//   DUTs/IO/Topology/ Beckhoff_AMI8xxxEK1122_B38FD36B.TcDUT (not stored), EK1100_Beckhoff_AMI8xxx_4205BDB3.TcDUT (not stored), EtherCAT_Master_AMIxxxx_FECF87C2.TcDUT (not stored), Beckhoff_APS1xxxEK1122_85E711A3.TcDUT (not stored), Beckhoff_APS1xxx_0455F8D3.TcDUT (not stored), Beckhoff_APS4xxxEK1122_65CE088F.TcDUT (not stored), Beckhoff_APS4xxx_87463DAF.TcDUT (not stored), EtherCAT_Master_APSxxxx_6FACD001.TcDUT (not stored), A_0060_AT2020_0250_0019_AT2020_0250_DEA07AF9.TcDUT (not stored), A_0036_AT2040_0250_0021_A3885EBC.TcDUT (not stored), A_0037_AT2040_0250_0022_971D272D.TcDUT (not stored), A_0038_AT2040_0250_0023_2AEAC7B2.TcDUT (not stored), A_0039_AT2040_0250_0024_A0FBBBF9.TcDUT (not stored), A_0040_AT2041_0250_0018_599416E0.TcDUT (not stored), A_0041_AT2041_0250_0019_45B99D70.TcDUT (not stored), A_0042_AT2041_0250_0020_B304CC62.TcDUT (not stored), A_0043_AT2041_0250_0021_3915B029.TcDUT (not stored), A_0044_AT2041_0250_0022_EA8B7A1C.TcDUT (not stored), A_0045_AT2041_0250_0023_5C753B73.TcDUT (not stored), A_0046_AT2042_0250_0024_35EBD522.TcDUT (not stored), A_0047_AT2050_0500_0016_017EACB3.TcDUT (not stored), A_0048_AT2050_0500_0017_A8B58F1D.TcDUT (not stored), A_0049_AT2050_0500_0018_A5979C2D.TcDUT (not stored), A_0050_AT2050_0500_0019_E6F81550.TcDUT (not stored), A_0051_AT2050_0500_0020_6A24DD88.TcDUT (not stored), A_0052_AT2050_0500_0021_294B54F5.TcDUT (not stored), A_0053_AT2050_0500_0022_49FE826D.TcDUT (not stored), A_0054_AT2050_0500_0023_9DD4EAFB.TcDUT (not stored), A_0055_AT2050_0500_0024_F6D8BACC.TcDUT (not stored), A_0056_AT2050_0501_0017_5F139962.TcDUT (not stored), A_0057_AT2050_0501_0020_6B86E0F3.TcDUT (not stored), A_0058_AT2050_0501_0021_54B106B2.TcDUT (not stored), A_0061_AT2020_0250_0023_AT2020_0250_0F2EDFD4.TcDUT (not stored), A_0062_AT2025_0250_0020_AT2025_0250_13035444.TcDUT (not stored), A_0063_AT2025_0250_0022_AT2025_0250_9D18840C.TcDUT (not stored), A_0064_AT2025_0250_0023_AT2025_0250_4A8CE23A.TcDUT (not stored), A_0065_AT2026_0250_0019_AT2026_0250_E347C194.TcDUT (not stored), A_0066_AT2026_0250_0020_AT2026_0250_D7D2B805.TcDUT (not stored), A_0067_AT2026_0250_0022_AT2026_0250_D02FEC70.TcDUT (not stored), A_0068_AT2026_0250_0024_AT2026_0250_BF201DA5.TcDUT (not stored), A_0069_AT2050_0501_0019_AT2050_0501_0D0F91BF.TcDUT (not stored), A_0070_AT2050_0501_0022_AT2050_0501_871EEDF4.TcDUT (not stored), A_0071_AT2050_0501_0023_AT2050_0501_6B46D2C7.TcDUT (not stored), A_0072_AT2050_0501_0024_AT2050_0501_776B5957.TcDUT (not stored), Beckhoff_AT2xxxEK1122_56C52038.TcDUT (not stored), Beckhoff_AT1xxx_7510A45A.TcDUT (not stored), A_0001_ATH2000_0250_0022_20236C4E.TcDUT (not stored), A_0002_ATH2000_0250_0023_D700A2ED.TcDUT (not stored), Beckhoff_ATH2xxxEK1122_13FBDC00.TcDUT (not stored), Beckhoff_ATH2xxx_159CB27D.TcDUT (not stored), EtherCAT_Master_ATxxxx_83672136.TcDUT (not stored), Beckhoff_AX2xxxEK1122_5FAF3C40.TcDUT (not stored), Beckhoff_AX2xxx_B0467A4D.TcDUT (not stored), Beckhoff_AX5xxxEK1122_5EFAAD43.TcDUT (not stored), Beckhoff_AX5xxx_ABA3CB51.TcDUT (not stored), Beckhoff_AX8yxxEK1122_5DB842B3.TcDUT (not stored), Beckhoff_AX8yxx_9373B1FA.TcDUT (not stored), Beckhoff_AX86xxEK1122_9E61CBD7.TcDUT (not stored), Beckhoff_AX86xx_1E3C21C9.TcDUT (not stored), Beckhoff_AX88xxEK1122_27E1F918.TcDUT (not stored), Beckhoff_AX88xx_5781E6BD.TcDUT (not stored), EtherCAT_Master_AXxxxx_5BD89A80.TcDUT (not stored), A_0014_BK1250_0000_0000_A4796D49.TcDUT (not stored), Beckhoff_BKxxxxsub_EK1100_CE1F4926.TcDUT (not stored), A_0001_BK1120_0000_0000_A11D37A6.TcDUT (not stored), A_0002_BK1120_0000_0001_6C916313.TcDUT (not stored), A_0003_BK1120_0000_0016_3EC4837B.TcDUT (not stored), A_0004_BK1120_0000_0017_F348D7CE.TcDUT (not stored), A_0005_BK1120_0000_0018_EC8BABB1.TcDUT (not stored), A_0006_BK1120_0000_0019_2107FF04.TcDUT (not stored), A_0007_BK1120_0000_0020_2D4D5A66.TcDUT (not stored), A_0008_BK1120_0000_0021_E0C10ED3.TcDUT (not stored), A_0009_CPXXXX_BK1150_0016_B294EEBB.TcDUT (not stored), A_0010_BK1150_0000_0016_7F18BA0E.TcDUT (not stored), A_0011_BK1150_0000_0017_163F2E6B.TcDUT (not stored), A_0012_BK1150_0000_0018_DBB37ADE.TcDUT (not stored), A_0013_BK1150_0000_0019_89E69AB6.TcDUT (not stored), A_0016_BK1250_0000_0017_446ACE03.TcDUT (not stored), Term_474_EK1100_44DC070B.TcDUT (not stored), A_0018_BK1250_0000_0019_5BA9B27C.TcDUT (not stored), Term_476_EK1100_ED4AD6ED.TcDUT (not stored), A_0017_BK1250_0000_0018_9625E6C9.TcDUT (not stored), Term_478_EK1100_69E708A2.TcDUT (not stored), A_0019_IL2300_B110_0016_D7C567E6.TcDUT (not stored), A_0020_IL2300_B110_0017_5C3C5D52.TcDUT (not stored), A_0021_IL2301_B110_0016_18E5DAA8.TcDUT (not stored), A_0022_IL2301_B110_0017_CE2B414F.TcDUT (not stored), A_0023_IL2302_B110_0016_9156D55C.TcDUT (not stored), A_0024_IL2302_B110_0017_7CD378DF.TcDUT (not stored), Beckhoff_BKxxxxEK1122_F2DB5C09.TcDUT (not stored), A_0015_BK1250_0000_0016_69F539FC.TcDUT (not stored), Beckhoff_BKxxxx_655B2331.TcDUT (not stored), A_0006_CU1128_0000_0002_0DB5F5B9.TcDUT (not stored), A_0005_CU1128_0000_0001_15602991.TcDUT (not stored), A_0004_CU1128_0000_0000_E069C544.TcDUT (not stored), A_0003_CU1124_0000_0016_F6CF179A.TcDUT (not stored), A_0002_CU1123_0010_0016_C16CD0B3.TcDUT (not stored), A_0001_CU1123_0000_0016_A8E4CC63.TcDUT (not stored), Beckhoff_CUxxxxEK1122_8084EAF6.TcDUT (not stored), Beckhoff_CUxxxx_D57B3A25.TcDUT (not stored), Beckhoff_CXxxxxEK1122_6E1B70A9.TcDUT (not stored), Beckhoff_CXxxxx_5AB893DE.TcDUT (not stored), TcTerminals210_1BK1250_5A51D777.TcDUT (not stored), TcTerminals210_EK1100_1_99191ECD.TcDUT (not stored), TcTerminals210_2BK1250_08988889.TcDUT (not stored), TcTerminals210_EK1100_2_BDAFA3B6.TcDUT (not stored), EtherCAT_Master_BKCUCX_8F70BCEA.TcDUT (not stored), Beckhoff_EJ1xxxEK1122_5D41058A.TcDUT (not stored), Beckhoff_EJ1xxx_BA4DEDCC.TcDUT (not stored), Beckhoff_EJ2xxxEK1122_7BCCD4D9.TcDUT (not stored), Beckhoff_EJ2xxx_42F4B05B.TcDUT (not stored), Beckhoff_EJ3xxxEK1122_6922078E.TcDUT (not stored), Beckhoff_EJ3xxx_E0C24C98.TcDUT (not stored), Beckhoff_EJ4xxxEK1122_15AA3F2B.TcDUT (not stored), Beckhoff_EJ4xxx_B433EAC7.TcDUT (not stored), Beckhoff_EJ5xxxEK1122_0744EC7C.TcDUT (not stored), Beckhoff_EJ5xxx_DF22D5A3.TcDUT (not stored), Beckhoff_EJ6xxxEK1122_30779985.TcDUT (not stored), Beckhoff_EJ6xxx_A0E5C2C0.TcDUT (not stored), Beckhoff_EJ7xxxEK1122_22994AD2.TcDUT (not stored), Beckhoff_EJ7xxx_9F75012E.TcDUT (not stored), Beckhoff_EJ9xxxEK1122_DB893B98.TcDUT (not stored), Beckhoff_EJ9xxx_660B2C8D.TcDUT (not stored), Beckhoff_EJx9xxEK1122_05D2B413.TcDUT (not stored), Beckhoff_EJx9xx_A9128509.TcDUT (not stored), EtherCAT_Master_EJxxxx_A1D13F1B.TcDUT (not stored), Beckhoff_EK11xxEK1122_0F9A1885.TcDUT (not stored), Beckhoff_EK11xx_C12453FF.TcDUT (not stored), Beckhoff_EK12xxEK1122_E9998301.TcDUT (not stored), Beckhoff_EK12xx_26FD3E4A.TcDUT (not stored), Beckhoff_EK13xxEK1122_7883D180.TcDUT (not stored), Beckhoff_EK13xx_F78FC0F8.TcDUT (not stored), Beckhoff_EK15xxEK1122_F4825052.TcDUT (not stored), Beckhoff_EK15xx_2CCE234B.TcDUT (not stored), Beckhoff_EK18xxEK1122_46BB19D8.TcDUT (not stored), Beckhoff_EK18xx_2BB31392.TcDUT (not stored), Beckhoff_EKM1xxxEK1122_D80A806C.TcDUT (not stored), Beckhoff_EKM1xxx_4291A3D4.TcDUT (not stored), Beckhoff_EKx9xxEK1122_199990A5.TcDUT (not stored), Beckhoff_EKx9xx_14304971.TcDUT (not stored), Beckhoff_EKxxxx_0080EK1122_49C116CC.TcDUT (not stored), Beckhoff_EKxxxx_0080_F8E2E0BC.TcDUT (not stored), EtherCAT_Master_EKxxxx_AFFC15C4.TcDUT (not stored), Beckhoff_ELM3xxxEK1122_52A3E13B.TcDUT (not stored), Beckhoff_ELM3xxx_6EC4C133.TcDUT (not stored), Beckhoff_ELM31xxEK1122_3E17608C.TcDUT (not stored), Beckhoff_ELM31xx_1B5DD775.TcDUT (not stored), Beckhoff_ELM35xxEK1122_B82F516C.TcDUT (not stored), Beckhoff_ELM35xx_45F1AC79.TcDUT (not stored), Beckhoff_ELM36xxEK1122_DABD45E4.TcDUT (not stored), Beckhoff_ELM36xx_F5043D7C.TcDUT (not stored), Beckhoff_ELM37xxEK1122_FB33499C.TcDUT (not stored), Beckhoff_ELM37xx_37DB7D9A.TcDUT (not stored), Beckhoff_ELM3xxx_0030EK1122_7F195F23.TcDUT (not stored), Beckhoff_ELM3xxx_0030_86EC0720.TcDUT (not stored), Beckhoff_ELM9xxxEK1122_E008DD2D.TcDUT (not stored), Beckhoff_ELM9xxx_2CCFEFDC.TcDUT (not stored), EtherCAT_Master_ELMxxxx_F3377F79.TcDUT (not stored), Beckhoff_EL1xxxEK1122_BA3F35BD.TcDUT (not stored), Beckhoff_EL1xxx_A02C084E.TcDUT (not stored), Beckhoff_EL2xxxEK1122_8D0C4044.TcDUT (not stored), Beckhoff_EL2xxx_6D51086F.TcDUT (not stored), Beckhoff_EL3xxxEK1122_9FE29313.TcDUT (not stored), Beckhoff_EL3xxx_68884AC1.TcDUT (not stored), Beckhoff_EL3xxx_0030EK1122_A8C7E601.TcDUT (not stored), Beckhoff_EL3xxx_0030_2D07FB6C.TcDUT (not stored), Beckhoff_EL4xxxEK1122_E36AABB6.TcDUT (not stored), Beckhoff_EL4xxx_B43A2050.TcDUT (not stored), Beckhoff_EL5xxxEK1122_F18478E1.TcDUT (not stored), Beckhoff_EL5xxx_C80BAEFE.TcDUT (not stored), Beckhoff_EL6xxxEK1122_C6B70D18.TcDUT (not stored), Beckhoff_EL6xxx_F14D3E2E.TcDUT (not stored), Beckhoff_EL7xxxEK1122_D459DE4F.TcDUT (not stored), Beckhoff_EL7xxx_9130E37B.TcDUT (not stored), Beckhoff_EL9xxxEK1122_2D49AF05.TcDUT (not stored), Beckhoff_EL9xxx_842928EF.TcDUT (not stored), Beckhoff_EL15xxEK1122_50B385EA.TcDUT (not stored), Beckhoff_EL15xx_DB59F57A.TcDUT (not stored), Beckhoff_EL19xxEK1122_DE3ACA7D.TcDUT (not stored), Beckhoff_EL19xx_39A0946F.TcDUT (not stored), Beckhoff_EL25xxEK1122_6780F013.TcDUT (not stored), Beckhoff_EL25xx_19393863.TcDUT (not stored), Beckhoff_EL29xxEK1122_E909BF84.TcDUT (not stored), Beckhoff_EL29xx_4C00A64E.TcDUT (not stored), Beckhoff_EL30xxEK1122_D2D81EDC.TcDUT (not stored), Beckhoff_EL30xx_21D80093.TcDUT (not stored), Beckhoff_EL31xxEK1122_F35612A4.TcDUT (not stored), Beckhoff_EL31xx_0F318B7E.TcDUT (not stored), Beckhoff_EL32xxEK1122_91C4062C.TcDUT (not stored), Beckhoff_EL32xx_64999344.TcDUT (not stored), Beckhoff_EL33xxEK1122_B04A0A54.TcDUT (not stored), Beckhoff_EL33xx_B84F5D38.TcDUT (not stored), Beckhoff_EL34xxEK1122_54E02F3C.TcDUT (not stored), Beckhoff_EL34xx_4C2EC3D0.TcDUT (not stored), Beckhoff_EL37xxEK1122_36723BB4.TcDUT (not stored), Beckhoff_EL37xx_735867E2.TcDUT (not stored), Beckhoff_EL47xxEK1122_4AFA0311.TcDUT (not stored), Beckhoff_EL47xx_965E5194.TcDUT (not stored), Beckhoff_EL66xxEK1122_D63A030B.TcDUT (not stored), Beckhoff_EL66xx_C1E1F370.TcDUT (not stored), Beckhoff_EL67xxEK1122_6F27A5BF.TcDUT (not stored), Beckhoff_EL67xx_2DE66D45.TcDUT (not stored), Beckhoff_EL68xxEK1122_833CFEA0.TcDUT (not stored), Beckhoff_EL68xx_2DEB682D.TcDUT (not stored), Beckhoff_EL69xxEK1122_A2B2F2D8.TcDUT (not stored), Beckhoff_EL69xx_A41E2827.TcDUT (not stored), Beckhoff_EL72xxEK1122_DA7F4B70.TcDUT (not stored), Beckhoff_EL72xx_B1894506.TcDUT (not stored), Beckhoff_EL73xxEK1122_FBF14708.TcDUT (not stored), Beckhoff_EL73xx_9CF0DC04.TcDUT (not stored), Beckhoff_EL99xxEK1122_494C50C5.TcDUT (not stored), A_0003_EL9930_0000_0017_255119B7.TcDUT (not stored), A_0001_EL9930_0000_0016_8200DBB0.TcDUT (not stored), Beckhoff_EL99xx_E89A1FE1.TcDUT (not stored), EtherCAT_Master_ELxxxx_D51EE2EF.TcDUT (not stored), Beckhoff_ELXxxxxEK1122_CE175A58.TcDUT (not stored), Beckhoff_ELXxxxx_091FCA88.TcDUT (not stored), EtherCAT_Master_ELXxxxx_037A66B5.TcDUT (not stored), Beckhoff_EM2xxxEK1122_264CF75A.TcDUT (not stored), Beckhoff_EM2xxx_D8CD5456.TcDUT (not stored), Beckhoff_EM3xxxEK1122_34A2240D.TcDUT (not stored), Beckhoff_EM3xxx_0E1B0655.TcDUT (not stored), Beckhoff_EM7xxxEK1122_7F196951.TcDUT (not stored), Beckhoff_EM7xxx_B71DC934.TcDUT (not stored), EtherCAT_Master_EMxxxx_4F6AEAF3.TcDUT (not stored), A_0024_EPP1342_0001_0017_B861A008.TcDUT (not stored), A_0023_EPP1342_0001_0016_F32E5EF0.TcDUT (not stored), A_0022_EPP1332_0001_0017_4E5F00D5.TcDUT (not stored), A_0021_EPP1332_0001_0016_0C75CF60.TcDUT (not stored), A_0020_EPP1322_0001_0017_AE45DA7A.TcDUT (not stored), A_0019_EPP1322_0001_0016_1D230593.TcDUT (not stored), A_0018_EPP1321_0060_0016_CF61AE2B.TcDUT (not stored), Beckhoff_EPP1xxxEK1122_CF9B9B85.TcDUT (not stored), Beckhoff_EPP1xxx_9DC54301.TcDUT (not stored), Beckhoff_EPP2xxxEK1122_0CAC7812.TcDUT (not stored), Beckhoff_EPP2xxx_7FE046AD.TcDUT (not stored), Beckhoff_EPP3xxxEK1122_936585F9.TcDUT (not stored), Beckhoff_EPP3xxx_5AF4C5F1.TcDUT (not stored), Beckhoff_EPP4xxxEK1122_A96F30AF.TcDUT (not stored), Beckhoff_EPP4xxx_454DDD33.TcDUT (not stored), Beckhoff_EPP5xxxEK1122_277DA9AB.TcDUT (not stored), Beckhoff_EPP5xxx_36D2ADAB.TcDUT (not stored), Beckhoff_EPP6xxxEK1122_580439A8.TcDUT (not stored), Beckhoff_EPP6xxx_5B035970.TcDUT (not stored), Beckhoff_EPP7xxxEK1122_0D11CA3B.TcDUT (not stored), Beckhoff_EPP7xxx_19C1DAAF.TcDUT (not stored), Beckhoff_EPP9xxxEK1122_5167694C.TcDUT (not stored), Beckhoff_EPP9xxx_B13825D2.TcDUT (not stored), EtherCAT_Master_EPPxxxx_7CC0E3EC.TcDUT (not stored), A_0037_EP1312_0001_0016_91E425AA.TcDUT (not stored), A_0026_EP1122_0001_0018_C0E43096.TcDUT (not stored), A_0025_EP1122_0001_0017_02B37791.TcDUT (not stored), A_0024_EP1122_0001_0016_1C40CD3A.TcDUT (not stored), Beckhoff_EP1xxxEK1122_B7B20563.TcDUT (not stored), Beckhoff_EP1xxx_C8E7C95B.TcDUT (not stored), Beckhoff_EP2xxxEK1122_CF43FCA1.TcDUT (not stored), Beckhoff_EP2xxx_B2F46B5A.TcDUT (not stored), Beckhoff_EP3xxxEK1122_961F7095.TcDUT (not stored), Beckhoff_EP3xxx_2B029919.TcDUT (not stored), Beckhoff_EP4xxxEK1122_BB643D5B.TcDUT (not stored), Beckhoff_EP4xxx_3DB4D53F.TcDUT (not stored), Beckhoff_EP5xxxEK1122_41313438.TcDUT (not stored), Beckhoff_EP5xxx_8FA7D670.TcDUT (not stored), Beckhoff_EP6xxxEK1122_E79FCD0D.TcDUT (not stored), Beckhoff_EP6xxx_66B3A0F3.TcDUT (not stored), A_0054_EP7402_0057_0017_54490F59.TcDUT (not stored), Beckhoff_EP7xxxEK1122_A7CCCB3C.TcDUT (not stored), Beckhoff_EP7xxx_5B32BB7C.TcDUT (not stored), Beckhoff_EP8xxxEK1122_09026D55.TcDUT (not stored), Beckhoff_EP8xxx_A1F98A04.TcDUT (not stored), A_0024_EP9521_0020_0000_2C408F2A.TcDUT (not stored), A_0022_EP9224_0037_0017_E33DE408.TcDUT (not stored), A_0013_EP9128_0021_0019_07EDD1EA.TcDUT (not stored), A_0010_EP9128_0021_0018_A4E84267.TcDUT (not stored), A_0007_EP9128_0021_0017_0A93B569.TcDUT (not stored), A_0004_EP9128_0021_0016_B7B89D3D.TcDUT (not stored), A_0001_EP9128_0020_0016_7FD3BAFD.TcDUT (not stored), Beckhoff_EP9xxxEK1122_D439D8FD.TcDUT (not stored), Beckhoff_EP9xxx_40638FD6.TcDUT (not stored), EtherCAT_Master_EPxxxx_AD623DA0.TcDUT (not stored), Beckhoff_EQ1xxxEK1122_FDDE2AD8.TcDUT (not stored), Beckhoff_EQ1xxx_822DEADB.TcDUT (not stored), Beckhoff_EQ2xxxEK1122_609ED827.TcDUT (not stored), Beckhoff_EQ2xxx_ABA09D4F.TcDUT (not stored), Beckhoff_EQ3xxxEK1122_C2B88B71.TcDUT (not stored), Beckhoff_EQ3xxx_1BCF419C.TcDUT (not stored), EtherCAT_Master_EQxxxx_C1E8A49A.TcDUT (not stored), Beckhoff_ER1xxxEK1122_03B27612.TcDUT (not stored), Beckhoff_ER1xxx_F144525A.TcDUT (not stored), Beckhoff_ER2xxxEK1122_C26931CF.TcDUT (not stored), Beckhoff_ER2xxx_C2CD7B25.TcDUT (not stored), Beckhoff_ER3xxxEK1122_1C34A142.TcDUT (not stored), Beckhoff_ER3xxx_0B6E7FA9.TcDUT (not stored), Beckhoff_ER4xxxEK1122_D1435FD1.TcDUT (not stored), Beckhoff_ER4xxx_C7805EB0.TcDUT (not stored), Beckhoff_ER5xxxEK1122_8A557ABF.TcDUT (not stored), Beckhoff_ER5xxx_1B1665E3.TcDUT (not stored), Beckhoff_ER6xxxEK1122_7ED5D873.TcDUT (not stored), Beckhoff_ER6xxx_39EF444F.TcDUT (not stored), Beckhoff_ER7xxxEK1122_C27AB41B.TcDUT (not stored), Beckhoff_ER7xxx_A258BD7D.TcDUT (not stored), Beckhoff_ER8xxxEK1122_05C4D0D1.TcDUT (not stored), Beckhoff_ER8xxx_BCCF5157.TcDUT (not stored), EtherCAT_Master_ERxxxx_D3400E61.TcDUT (not stored), TcTerminals210_1EK1100_99191ECD.TcDUT (not stored), TcTerminals210_2EK1100_BDAFA3B6.TcDUT (not stored), EtherCAT_Master_KLxxxx_4E9397D5.TcDUT (not stored), EtherCAT_Master_KLxxxx_1_B89C6D7A.TcDUT (not stored), EtherCAT_Master_KLxxxx_2_C1BBE75B.TcDUT (not stored), boxesEK1122_6347E441.TcDUT (not stored), boxes_B14E9406.TcDUT (not stored), EtherCAT_Master_Duplicates_FF3295D1.TcDUT (not stored)
//   GVLs/ GVL_iXlinker.TcGVL

// ---- DUTs/IO/Boxes/EK1100_179A0949.TcDUT
{attribute addProperty BoxType "EK1100-0000-0018"}
{attribute addProperty Id "InfoDataInfoData_192954DE162"}
{attribute addProperty CRC "395970889"}
{attribute addProperty SizeInBites "16"}
{attribute addProperty SizeInBytes "2"}
TYPE EK1100_179A0949 :
STRUCT
	{attribute addProperty Name "InfoData"}
	InfoData : InfoData_192954DE;
END_STRUCT
END_TYPE

// ---- DUTs/IO/Boxes/EK1122_179A0949.TcDUT
{attribute addProperty BoxType "EK1122-0000-0018"}
{attribute addProperty Id "InfoDataInfoData_192954DE162"}
{attribute addProperty CRC "395970889"}
{attribute addProperty SizeInBites "16"}
{attribute addProperty SizeInBytes "2"}
TYPE EK1122_179A0949 :
STRUCT
	{attribute addProperty Name "InfoData"}
	InfoData : InfoData_192954DE;
END_STRUCT
END_TYPE

// ---- DUTs/IO/Boxes/AMI8000_17A3F7C1.TcDUT
{attribute addProperty BoxType "AMI8000-0000-0016"}
{attribute addProperty Id "FB_PositionAT %I*FB_Position_BA8AA9F03240DRV_StatuswordAT %I*DRV_Statusword_53CBCECC1620DRV_Following_error_actual_valueAT %I*DRV_Following_error_actual_value_F54335363240DRV_ControlwordAT %Q*DRV_Controlword_417617681620DRV_Target_positionAT %Q*DRV_Target_position_41334FAA3240WcStateAT %I*WcState_98A4DF7520.250InfoDataAT %I*InfoData_BF6E01EA168210"}
{attribute addProperty CRC "4025043701"}
{attribute addProperty SizeInBites "298"}
{attribute addProperty SizeInBytes "37.25"}
TYPE AMI8000_17A3F7C1 :
STRUCT
	{attribute addProperty Name "FB_Position"}
	FB_Position : FB_Position_BA8AA9F0;
	{attribute addProperty Name "DRV_Statusword"}
	DRV_Statusword : DRV_Statusword_53CBCECC;
	{attribute addProperty Name "DRV_Following_error_actual_value"}
	DRV_Following_error_actual_value : DRV_Following_error_actual_value_F5433536;
	{attribute addProperty Name "DRV_Controlword"}
	DRV_Controlword : DRV_Controlword_41761768;
	{attribute addProperty Name "DRV_Target_position"}
	DRV_Target_position : DRV_Target_position_41334FAA;
	{attribute addProperty Name "WcState"}
	WcState : WcState_98A4DF75;
	{attribute addProperty Name "InfoData"}
	InfoData : InfoData_BF6E01EA;
END_STRUCT
END_TYPE

// ---- DUTs/IO/Boxes/APS1003_D6441620.TcDUT
{attribute addProperty BoxType "APS1003-7000-0016"}
{attribute addProperty Id "YVR_InputsAT %I*YVR_Inputs_32B3017D784980YVR_OutputsAT %Q*YVR_Outputs_0CD1622111681460WcStateAT %I*WcState_98A4DF7520.250InfoDataAT %I*InfoData_0BDED7BF144180"}
{attribute addProperty CRC "271105188"}
{attribute addProperty SizeInBites "2098"}
{attribute addProperty SizeInBytes "262.25"}
TYPE APS1003_D6441620 :
STRUCT
	{attribute addProperty Name "YVR_Inputs"}
	YVR_Inputs : YVR_Inputs_32B3017D;
	{attribute addProperty Name "YVR_Outputs"}
	YVR_Outputs : YVR_Outputs_0CD16221;
	{attribute addProperty Name "WcState"}
	WcState : WcState_98A4DF75;
	{attribute addProperty Name "InfoData"}
	InfoData : InfoData_0BDED7BF;
END_STRUCT
END_TYPE

// ---- DUTs/IO/Boxes/APS1003_59AFCAF5.TcDUT
{attribute addProperty BoxType "APS1003-5000-0016"}
{attribute addProperty Id "FB_InputsAT %I*FB_Inputs_245CD1AC24643080WcStateAT %I*WcState_98A4DF7520.250InfoDataAT %I*InfoData_7231B2DD80100"}
{attribute addProperty CRC "2263788637"}
{attribute addProperty SizeInBites "2546"}
{attribute addProperty SizeInBytes "318.25"}
TYPE APS1003_59AFCAF5 :
STRUCT
	{attribute addProperty Name "FB_Inputs"}
	FB_Inputs : FB_Inputs_245CD1AC;
	{attribute addProperty Name "WcState"}
	WcState : WcState_98A4DF75;
	{attribute addProperty Name "InfoData"}
	InfoData : InfoData_7231B2DD;
END_STRUCT
END_TYPE

// ---- DUTs/IO/Boxes/APS4322_1E964C4E.TcDUT
{attribute addProperty BoxType "APS4322-7000-0017"}
{attribute addProperty Id "APS_InputsAT %I*APS_Inputs_32B3017D784980APS_DiagdataAT %I*APS_Diagdata_9B5B9C043240APS_Comm_InputsAT %I*APS_Comm_Inputs_FF1CE56E80100APS_OutputsAT %Q*APS_Outputs_0CD1622111681460APS_Comm_OutputsAT %Q*APS_Comm_Outputs_D1BECFC43240WcStateAT %I*WcState_98A4DF7520.250InfoDataAT %I*InfoData_0BDED7BF144180"}
{attribute addProperty CRC "1396157949"}
{attribute addProperty SizeInBites "2242"}
{attribute addProperty SizeInBytes "280.25"}
TYPE APS4322_1E964C4E :
STRUCT
	{attribute addProperty Name "APS_Inputs"}
	APS_Inputs : APS_Inputs_32B3017D;
	{attribute addProperty Name "APS_Diagdata"}
	APS_Diagdata : APS_Diagdata_9B5B9C04;
	{attribute addProperty Name "APS_Comm_Inputs"}
	APS_Comm_Inputs : APS_Comm_Inputs_FF1CE56E;
	{attribute addProperty Name "APS_Outputs"}
	APS_Outputs : APS_Outputs_0CD16221;
	{attribute addProperty Name "APS_Comm_Outputs"}
	APS_Comm_Outputs : APS_Comm_Outputs_D1BECFC4;
	{attribute addProperty Name "WcState"}
	WcState : WcState_98A4DF75;
	{attribute addProperty Name "InfoData"}
	InfoData : InfoData_0BDED7BF;
END_STRUCT
END_TYPE

// ---- DUTs/IO/Boxes/APS4322_59AFCAF5.TcDUT
{attribute addProperty BoxType "APS4322-5000-0017"}
{attribute addProperty Id "FB_InputsAT %I*FB_Inputs_245CD1AC24643080WcStateAT %I*WcState_98A4DF7520.250InfoDataAT %I*InfoData_7231B2DD80100"}
{attribute addProperty CRC "2263788637"}
{attribute addProperty SizeInBites "2546"}
{attribute addProperty SizeInBytes "318.25"}
TYPE APS4322_59AFCAF5 :
STRUCT
	{attribute addProperty Name "FB_Inputs"}
	FB_Inputs : FB_Inputs_245CD1AC;
	{attribute addProperty Name "WcState"}
	WcState : WcState_98A4DF75;
	{attribute addProperty Name "InfoData"}
	InfoData : InfoData_7231B2DD;
END_STRUCT
END_TYPE

// ---- DUTs/IO/Boxes/AT2020_BA5A9548.TcDUT
{attribute addProperty BoxType "AT2020-0250-0019"}
{attribute addProperty Id "CC_InputsAT %I*CC_Inputs_9818D8D8256320CC_OutputsAT %Q*CC_Outputs_AA78E99F256320WcStateAT %I*WcState_98A4DF7520.250InfoDataAT %I*InfoData_0BDED7BF144180"}
{attribute addProperty CRC "3298337665"}
{attribute addProperty SizeInBites "658"}
{attribute addProperty SizeInBytes "82.25"}
TYPE AT2020_BA5A9548 :
STRUCT
	{attribute addProperty Name "CC_Inputs"}
	CC_Inputs : CC_Inputs_9818D8D8;
	{attribute addProperty Name "CC_Outputs"}
	CC_Outputs : CC_Outputs_AA78E99F;
	{attribute addProperty Name "WcState"}
	WcState : WcState_98A4DF75;
	{attribute addProperty Name "InfoData"}
	InfoData : InfoData_0BDED7BF;
END_STRUCT
END_TYPE

// ---- DUTs/IO/Boxes/AT2050_C5E59848.TcDUT
{attribute addProperty BoxType "AT2050-5500-0018"}
{attribute addProperty Id "FB_InputsAT %I*FB_Inputs_A6E87AE0528660FB_OutputsAT %Q*FB_Outputs_734938A41620WcStateAT %I*WcState_98A4DF7520.250InfoDataAT %I*InfoData_7231B2DD80100"}
{attribute addProperty CRC "2967070852"}
{attribute addProperty SizeInBites "626"}
{attribute addProperty SizeInBytes "78.25"}
TYPE AT2050_C5E59848 :
STRUCT
	{attribute addProperty Name "FB_Inputs"}
	FB_Inputs : FB_Inputs_A6E87AE0;
	{attribute addProperty Name "FB_Outputs"}
	FB_Outputs : FB_Outputs_734938A4;
	{attribute addProperty Name "WcState"}
	WcState : WcState_98A4DF75;
	{attribute addProperty Name "InfoData"}
	InfoData : InfoData_7231B2DD;
END_STRUCT
END_TYPE

// ---- DUTs/IO/Boxes/AT2000_15405010.TcDUT
{attribute addProperty BoxType "AT2000-0233-0022"}
{attribute addProperty Id "CC_Inputs_14_ChAT %I*CC_Inputs_14_Ch_5FB71CBE240300CC_Outputs_14_ChAT %Q*CC_Outputs_14_Ch_8D55E481240300WcStateAT %I*WcState_98A4DF7520.250InfoDataAT %I*InfoData_0BDED7BF144180"}
{attribute addProperty CRC "2331747689"}
{attribute addProperty SizeInBites "626"}
{attribute addProperty SizeInBytes "78.25"}
TYPE AT2000_15405010 :
STRUCT
	{attribute addProperty Name "CC_Inputs_14_Ch"}
	CC_Inputs_14_Ch : CC_Inputs_14_Ch_5FB71CBE;
	{attribute addProperty Name "CC_Outputs_14_Ch"}
	CC_Outputs_14_Ch : CC_Outputs_14_Ch_8D55E481;
	{attribute addProperty Name "WcState"}
	WcState : WcState_98A4DF75;
	{attribute addProperty Name "InfoData"}
	InfoData : InfoData_0BDED7BF;
END_STRUCT
END_TYPE

// ---- DUTs/IO/Boxes/AT2000_BA5A9548.TcDUT
{attribute addProperty BoxType "AT2000-0250-0016"}
{attribute addProperty Id "CC_InputsAT %I*CC_Inputs_9818D8D8256320CC_OutputsAT %Q*CC_Outputs_AA78E99F256320WcStateAT %I*WcState_98A4DF7520.250InfoDataAT %I*InfoData_0BDED7BF144180"}
{attribute addProperty CRC "3298337665"}
{attribute addProperty SizeInBites "658"}
{attribute addProperty SizeInBytes "82.25"}
TYPE AT2000_BA5A9548 :
STRUCT
	{attribute addProperty Name "CC_Inputs"}
	CC_Inputs : CC_Inputs_9818D8D8;
	{attribute addProperty Name "CC_Outputs"}
	CC_Outputs : CC_Outputs_AA78E99F;
	{attribute addProperty Name "WcState"}
	WcState : WcState_98A4DF75;
	{attribute addProperty Name "InfoData"}
	InfoData : InfoData_0BDED7BF;
END_STRUCT
END_TYPE

// ---- DUTs/IO/Boxes/AT2001_BA5A9548.TcDUT
{attribute addProperty BoxType "AT2001-0250-0016"}
{attribute addProperty Id "CC_InputsAT %I*CC_Inputs_9818D8D8256320CC_OutputsAT %Q*CC_Outputs_AA78E99F256320WcStateAT %I*WcState_98A4DF7520.250InfoDataAT %I*InfoData_0BDED7BF144180"}
{attribute addProperty CRC "3298337665"}
{attribute addProperty SizeInBites "658"}
{attribute addProperty SizeInBytes "82.25"}
TYPE AT2001_BA5A9548 :
STRUCT
	{attribute addProperty Name "CC_Inputs"}
	CC_Inputs : CC_Inputs_9818D8D8;
	{attribute addProperty Name "CC_Outputs"}
	CC_Outputs : CC_Outputs_AA78E99F;
	{attribute addProperty Name "WcState"}
	WcState : WcState_98A4DF75;
	{attribute addProperty Name "InfoData"}
	InfoData : InfoData_0BDED7BF;
END_STRUCT
END_TYPE

// ---- DUTs/IO/Boxes/AT2002_BA5A9548.TcDUT
{attribute addProperty BoxType "AT2002-0249-0021"}
{attribute addProperty Id "CC_InputsAT %I*CC_Inputs_9818D8D8256320CC_OutputsAT %Q*CC_Outputs_AA78E99F256320WcStateAT %I*WcState_98A4DF7520.250InfoDataAT %I*InfoData_0BDED7BF144180"}
{attribute addProperty CRC "3298337665"}
{attribute addProperty SizeInBites "658"}
{attribute addProperty SizeInBytes "82.25"}
TYPE AT2002_BA5A9548 :
STRUCT
	{attribute addProperty Name "CC_Inputs"}
	CC_Inputs : CC_Inputs_9818D8D8;
	{attribute addProperty Name "CC_Outputs"}
	CC_Outputs : CC_Outputs_AA78E99F;
	{attribute addProperty Name "WcState"}
	WcState : WcState_98A4DF75;
	{attribute addProperty Name "InfoData"}
	InfoData : InfoData_0BDED7BF;
END_STRUCT
END_TYPE

// ---- DUTs/IO/Boxes/AT2021_BA5A9548.TcDUT
{attribute addProperty BoxType "AT2021-0250-0018"}
{attribute addProperty Id "CC_InputsAT %I*CC_Inputs_9818D8D8256320CC_OutputsAT %Q*CC_Outputs_AA78E99F256320WcStateAT %I*WcState_98A4DF7520.250InfoDataAT %I*InfoData_0BDED7BF144180"}
{attribute addProperty CRC "3298337665"}
{attribute addProperty SizeInBites "658"}
{attribute addProperty SizeInBytes "82.25"}
TYPE AT2021_BA5A9548 :
STRUCT
	{attribute addProperty Name "CC_Inputs"}
	CC_Inputs : CC_Inputs_9818D8D8;
	{attribute addProperty Name "CC_Outputs"}
	CC_Outputs : CC_Outputs_AA78E99F;
	{attribute addProperty Name "WcState"}
	WcState : WcState_98A4DF75;
	{attribute addProperty Name "InfoData"}
	InfoData : InfoData_0BDED7BF;
END_STRUCT
END_TYPE

// ---- DUTs/IO/Boxes/AT2025_BA5A9548.TcDUT
{attribute addProperty BoxType "AT2025-0250-0018"}
{attribute addProperty Id "CC_InputsAT %I*CC_Inputs_9818D8D8256320CC_OutputsAT %Q*CC_Outputs_AA78E99F256320WcStateAT %I*WcState_98A4DF7520.250InfoDataAT %I*InfoData_0BDED7BF144180"}
{attribute addProperty CRC "3298337665"}
{attribute addProperty SizeInBites "658"}
{attribute addProperty SizeInBytes "82.25"}
TYPE AT2025_BA5A9548 :
STRUCT
	{attribute addProperty Name "CC_Inputs"}
	CC_Inputs : CC_Inputs_9818D8D8;
	{attribute addProperty Name "CC_Outputs"}
	CC_Outputs : CC_Outputs_AA78E99F;
	{attribute addProperty Name "WcState"}
	WcState : WcState_98A4DF75;
	{attribute addProperty Name "InfoData"}
	InfoData : InfoData_0BDED7BF;
END_STRUCT
END_TYPE

// ---- DUTs/IO/Boxes/AT2026_BA5A9548.TcDUT
{attribute addProperty BoxType "AT2026-0250-0021"}
{attribute addProperty Id "CC_InputsAT %I*CC_Inputs_9818D8D8256320CC_OutputsAT %Q*CC_Outputs_AA78E99F256320WcStateAT %I*WcState_98A4DF7520.250InfoDataAT %I*InfoData_0BDED7BF144180"}
{attribute addProperty CRC "3298337665"}
{attribute addProperty SizeInBites "658"}
{attribute addProperty SizeInBytes "82.25"}
TYPE AT2026_BA5A9548 :
STRUCT
	{attribute addProperty Name "CC_Inputs"}
	CC_Inputs : CC_Inputs_9818D8D8;
	{attribute addProperty Name "CC_Outputs"}
	CC_Outputs : CC_Outputs_AA78E99F;
	{attribute addProperty Name "WcState"}
	WcState : WcState_98A4DF75;
	{attribute addProperty Name "InfoData"}
	InfoData : InfoData_0BDED7BF;
END_STRUCT
END_TYPE

// ---- DUTs/IO/Boxes/AT2040_BA5A9548.TcDUT
{attribute addProperty BoxType "AT2040-0250-0018"}
{attribute addProperty Id "CC_InputsAT %I*CC_Inputs_9818D8D8256320CC_OutputsAT %Q*CC_Outputs_AA78E99F256320WcStateAT %I*WcState_98A4DF7520.250InfoDataAT %I*InfoData_0BDED7BF144180"}
{attribute addProperty CRC "3298337665"}
{attribute addProperty SizeInBites "658"}
{attribute addProperty SizeInBytes "82.25"}
TYPE AT2040_BA5A9548 :
STRUCT
	{attribute addProperty Name "CC_Inputs"}
	CC_Inputs : CC_Inputs_9818D8D8;
	{attribute addProperty Name "CC_Outputs"}
	CC_Outputs : CC_Outputs_AA78E99F;
	{attribute addProperty Name "WcState"}
	WcState : WcState_98A4DF75;
	{attribute addProperty Name "InfoData"}
	InfoData : InfoData_0BDED7BF;
END_STRUCT
END_TYPE

// ---- DUTs/IO/Boxes/AT2000_C5E59848.TcDUT
{attribute addProperty BoxType "AT2000-5233-0019"}
{attribute addProperty Id "FB_InputsAT %I*FB_Inputs_A6E87AE0528660FB_OutputsAT %Q*FB_Outputs_734938A41620WcStateAT %I*WcState_98A4DF7520.250InfoDataAT %I*InfoData_7231B2DD80100"}
{attribute addProperty CRC "2967070852"}
{attribute addProperty SizeInBites "626"}
{attribute addProperty SizeInBytes "78.25"}
TYPE AT2000_C5E59848 :
STRUCT
	{attribute addProperty Name "FB_Inputs"}
	FB_Inputs : FB_Inputs_A6E87AE0;
	{attribute addProperty Name "FB_Outputs"}
	FB_Outputs : FB_Outputs_734938A4;
	{attribute addProperty Name "WcState"}
	WcState : WcState_98A4DF75;
	{attribute addProperty Name "InfoData"}
	InfoData : InfoData_7231B2DD;
END_STRUCT
END_TYPE

// ---- DUTs/IO/Boxes/AT2026_C5E59848.TcDUT
{attribute addProperty BoxType "AT2026-5250-0019"}
{attribute addProperty Id "FB_InputsAT %I*FB_Inputs_A6E87AE0528660FB_OutputsAT %Q*FB_Outputs_734938A41620WcStateAT %I*WcState_98A4DF7520.250InfoDataAT %I*InfoData_7231B2DD80100"}
{attribute addProperty CRC "2967070852"}
{attribute addProperty SizeInBites "626"}
{attribute addProperty SizeInBytes "78.25"}
TYPE AT2026_C5E59848 :
STRUCT
	{attribute addProperty Name "FB_Inputs"}
	FB_Inputs : FB_Inputs_A6E87AE0;
	{attribute addProperty Name "FB_Outputs"}
	FB_Outputs : FB_Outputs_734938A4;
	{attribute addProperty Name "WcState"}
	WcState : WcState_98A4DF75;
	{attribute addProperty Name "InfoData"}
	InfoData : InfoData_7231B2DD;
END_STRUCT
END_TYPE

// ---- DUTs/IO/Boxes/AT2041_BA5A9548.TcDUT
{attribute addProperty BoxType "AT2041-0250-0018"}
{attribute addProperty Id "CC_InputsAT %I*CC_Inputs_9818D8D8256320CC_OutputsAT %Q*CC_Outputs_AA78E99F256320WcStateAT %I*WcState_98A4DF7520.250InfoDataAT %I*InfoData_0BDED7BF144180"}
{attribute addProperty CRC "3298337665"}
{attribute addProperty SizeInBites "658"}
{attribute addProperty SizeInBytes "82.25"}
TYPE AT2041_BA5A9548 :
STRUCT
	{attribute addProperty Name "CC_Inputs"}
	CC_Inputs : CC_Inputs_9818D8D8;
	{attribute addProperty Name "CC_Outputs"}
	CC_Outputs : CC_Outputs_AA78E99F;
	{attribute addProperty Name "WcState"}
	WcState : WcState_98A4DF75;
	{attribute addProperty Name "InfoData"}
	InfoData : InfoData_0BDED7BF;
END_STRUCT
END_TYPE

// ---- DUTs/IO/Boxes/AT2042_C5E59848.TcDUT
{attribute addProperty BoxType "AT2042-5250-0019"}
{attribute addProperty Id "FB_InputsAT %I*FB_Inputs_A6E87AE0528660FB_OutputsAT %Q*FB_Outputs_734938A41620WcStateAT %I*WcState_98A4DF7520.250InfoDataAT %I*InfoData_7231B2DD80100"}
{attribute addProperty CRC "2967070852"}
{attribute addProperty SizeInBites "626"}
{attribute addProperty SizeInBytes "78.25"}
TYPE AT2042_C5E59848 :
STRUCT
	{attribute addProperty Name "FB_Inputs"}
	FB_Inputs : FB_Inputs_A6E87AE0;
	{attribute addProperty Name "FB_Outputs"}
	FB_Outputs : FB_Outputs_734938A4;
	{attribute addProperty Name "WcState"}
	WcState : WcState_98A4DF75;
	{attribute addProperty Name "InfoData"}
	InfoData : InfoData_7231B2DD;
END_STRUCT
END_TYPE

// ---- DUTs/IO/Boxes/AT2041_C5E59848.TcDUT
{attribute addProperty BoxType "AT2041-5250-0019"}
{attribute addProperty Id "FB_InputsAT %I*FB_Inputs_A6E87AE0528660FB_OutputsAT %Q*FB_Outputs_734938A41620WcStateAT %I*WcState_98A4DF7520.250InfoDataAT %I*InfoData_7231B2DD80100"}
{attribute addProperty CRC "2967070852"}
{attribute addProperty SizeInBites "626"}
{attribute addProperty SizeInBytes "78.25"}
TYPE AT2041_C5E59848 :
STRUCT
	{attribute addProperty Name "FB_Inputs"}
	FB_Inputs : FB_Inputs_A6E87AE0;
	{attribute addProperty Name "FB_Outputs"}
	FB_Outputs : FB_Outputs_734938A4;
	{attribute addProperty Name "WcState"}
	WcState : WcState_98A4DF75;
	{attribute addProperty Name "InfoData"}
	InfoData : InfoData_7231B2DD;
END_STRUCT
END_TYPE

// ---- DUTs/IO/Boxes/AT2040_C5E59848.TcDUT
{attribute addProperty BoxType "AT2040-5250-0019"}
{attribute addProperty Id "FB_InputsAT %I*FB_Inputs_A6E87AE0528660FB_OutputsAT %Q*FB_Outputs_734938A41620WcStateAT %I*WcState_98A4DF7520.250InfoDataAT %I*InfoData_7231B2DD80100"}
{attribute addProperty CRC "2967070852"}
{attribute addProperty SizeInBites "626"}
{attribute addProperty SizeInBytes "78.25"}
TYPE AT2040_C5E59848 :
STRUCT
	{attribute addProperty Name "FB_Inputs"}
	FB_Inputs : FB_Inputs_A6E87AE0;
	{attribute addProperty Name "FB_Outputs"}
	FB_Outputs : FB_Outputs_734938A4;
	{attribute addProperty Name "WcState"}
	WcState : WcState_98A4DF75;
	{attribute addProperty Name "InfoData"}
	InfoData : InfoData_7231B2DD;
END_STRUCT
END_TYPE

// ---- DUTs/IO/Boxes/AT2042_BA5A9548.TcDUT
{attribute addProperty BoxType "AT2042-0250-0024"}
{attribute addProperty Id "CC_InputsAT %I*CC_Inputs_9818D8D8256320CC_OutputsAT %Q*CC_Outputs_AA78E99F256320WcStateAT %I*WcState_98A4DF7520.250InfoDataAT %I*InfoData_0BDED7BF144180"}
{attribute addProperty CRC "3298337665"}
{attribute addProperty SizeInBites "658"}
{attribute addProperty SizeInBytes "82.25"}
TYPE AT2042_BA5A9548 :
STRUCT
	{attribute addProperty Name "CC_Inputs"}
	CC_Inputs : CC_Inputs_9818D8D8;
	{attribute addProperty Name "CC_Outputs"}
	CC_Outputs : CC_Outputs_AA78E99F;
	{attribute addProperty Name "WcState"}
	WcState : WcState_98A4DF75;
	{attribute addProperty Name "InfoData"}
	InfoData : InfoData_0BDED7BF;
END_STRUCT
END_TYPE

// ---- DUTs/IO/Boxes/AT2025_C5E59848.TcDUT
{attribute addProperty BoxType "AT2025-5250-0019"}
{attribute addProperty Id "FB_InputsAT %I*FB_Inputs_A6E87AE0528660FB_OutputsAT %Q*FB_Outputs_734938A41620WcStateAT %I*WcState_98A4DF7520.250InfoDataAT %I*InfoData_7231B2DD80100"}
{attribute addProperty CRC "2967070852"}
{attribute addProperty SizeInBites "626"}
{attribute addProperty SizeInBytes "78.25"}
TYPE AT2025_C5E59848 :
STRUCT
	{attribute addProperty Name "FB_Inputs"}
	FB_Inputs : FB_Inputs_A6E87AE0;
	{attribute addProperty Name "FB_Outputs"}
	FB_Outputs : FB_Outputs_734938A4;
	{attribute addProperty Name "WcState"}
	WcState : WcState_98A4DF75;
	{attribute addProperty Name "InfoData"}
	InfoData : InfoData_7231B2DD;
END_STRUCT
END_TYPE

// ---- DUTs/IO/Boxes/AT2050_BA5A9548.TcDUT
{attribute addProperty BoxType "AT2050-0500-0016"}
{attribute addProperty Id "CC_InputsAT %I*CC_Inputs_9818D8D8256320CC_OutputsAT %Q*CC_Outputs_AA78E99F256320WcStateAT %I*WcState_98A4DF7520.250InfoDataAT %I*InfoData_0BDED7BF144180"}
{attribute addProperty CRC "3298337665"}
{attribute addProperty SizeInBites "658"}
{attribute addProperty SizeInBytes "82.25"}
TYPE AT2050_BA5A9548 :
STRUCT
	{attribute addProperty Name "CC_Inputs"}
	CC_Inputs : CC_Inputs_9818D8D8;
	{attribute addProperty Name "CC_Outputs"}
	CC_Outputs : CC_Outputs_AA78E99F;
	{attribute addProperty Name "WcState"}
	WcState : WcState_98A4DF75;
	{attribute addProperty Name "InfoData"}
	InfoData : InfoData_0BDED7BF;
END_STRUCT
END_TYPE

// ---- DUTs/IO/Boxes/AT2021_C5E59848.TcDUT
{attribute addProperty BoxType "AT2021-5250-0019"}
{attribute addProperty Id "FB_InputsAT %I*FB_Inputs_A6E87AE0528660FB_OutputsAT %Q*FB_Outputs_734938A41620WcStateAT %I*WcState_98A4DF7520.250InfoDataAT %I*InfoData_7231B2DD80100"}
{attribute addProperty CRC "2967070852"}
{attribute addProperty SizeInBites "626"}
{attribute addProperty SizeInBytes "78.25"}
TYPE AT2021_C5E59848 :
STRUCT
	{attribute addProperty Name "FB_Inputs"}
	FB_Inputs : FB_Inputs_A6E87AE0;
	{attribute addProperty Name "FB_Outputs"}
	FB_Outputs : FB_Outputs_734938A4;
	{attribute addProperty Name "WcState"}
	WcState : WcState_98A4DF75;
	{attribute addProperty Name "InfoData"}
	InfoData : InfoData_7231B2DD;
END_STRUCT
END_TYPE

// ---- DUTs/IO/Boxes/AT2020_C5E59848.TcDUT
{attribute addProperty BoxType "AT2020-5250-0019"}
{attribute addProperty Id "FB_InputsAT %I*FB_Inputs_A6E87AE0528660FB_OutputsAT %Q*FB_Outputs_734938A41620WcStateAT %I*WcState_98A4DF7520.250InfoDataAT %I*InfoData_7231B2DD80100"}
{attribute addProperty CRC "2967070852"}
{attribute addProperty SizeInBites "626"}
{attribute addProperty SizeInBytes "78.25"}
TYPE AT2020_C5E59848 :
STRUCT
	{attribute addProperty Name "FB_Inputs"}
	FB_Inputs : FB_Inputs_A6E87AE0;
	{attribute addProperty Name "FB_Outputs"}
	FB_Outputs : FB_Outputs_734938A4;
	{attribute addProperty Name "WcState"}
	WcState : WcState_98A4DF75;
	{attribute addProperty Name "InfoData"}
	InfoData : InfoData_7231B2DD;
END_STRUCT
END_TYPE

// ---- DUTs/IO/Boxes/AT2001_C5E59848.TcDUT
{attribute addProperty BoxType "AT2001-5250-0017"}
{attribute addProperty Id "FB_InputsAT %I*FB_Inputs_A6E87AE0528660FB_OutputsAT %Q*FB_Outputs_734938A41620WcStateAT %I*WcState_98A4DF7520.250InfoDataAT %I*InfoData_7231B2DD80100"}
{attribute addProperty CRC "2967070852"}
{attribute addProperty SizeInBites "626"}
{attribute addProperty SizeInBytes "78.25"}
TYPE AT2001_C5E59848 :
STRUCT
	{attribute addProperty Name "FB_Inputs"}
	FB_Inputs : FB_Inputs_A6E87AE0;
	{attribute addProperty Name "FB_Outputs"}
	FB_Outputs : FB_Outputs_734938A4;
	{attribute addProperty Name "WcState"}
	WcState : WcState_98A4DF75;
	{attribute addProperty Name "InfoData"}
	InfoData : InfoData_7231B2DD;
END_STRUCT
END_TYPE

// ---- DUTs/IO/Boxes/AT2002_C5E59848.TcDUT
{attribute addProperty BoxType "AT2002-5249-0018"}
{attribute addProperty Id "FB_InputsAT %I*FB_Inputs_A6E87AE0528660FB_OutputsAT %Q*FB_Outputs_734938A41620WcStateAT %I*WcState_98A4DF7520.250InfoDataAT %I*InfoData_7231B2DD80100"}
{attribute addProperty CRC "2967070852"}
{attribute addProperty SizeInBites "626"}
{attribute addProperty SizeInBytes "78.25"}
TYPE AT2002_C5E59848 :
STRUCT
	{attribute addProperty Name "FB_Inputs"}
	FB_Inputs : FB_Inputs_A6E87AE0;
	{attribute addProperty Name "FB_Outputs"}
	FB_Outputs : FB_Outputs_734938A4;
	{attribute addProperty Name "WcState"}
	WcState : WcState_98A4DF75;
	{attribute addProperty Name "InfoData"}
	InfoData : InfoData_7231B2DD;
END_STRUCT
END_TYPE

// ---- DUTs/IO/Boxes/ATH2000_BA5A9548.TcDUT
{attribute addProperty BoxType "ATH2000-0250-0022"}
{attribute addProperty Id "CC_InputsAT %I*CC_Inputs_9818D8D8256320CC_OutputsAT %Q*CC_Outputs_AA78E99F256320WcStateAT %I*WcState_98A4DF7520.250InfoDataAT %I*InfoData_0BDED7BF144180"}
{attribute addProperty CRC "3298337665"}
{attribute addProperty SizeInBites "658"}
{attribute addProperty SizeInBytes "82.25"}
TYPE ATH2000_BA5A9548 :
STRUCT
	{attribute addProperty Name "CC_Inputs"}
	CC_Inputs : CC_Inputs_9818D8D8;
	{attribute addProperty Name "CC_Outputs"}
	CC_Outputs : CC_Outputs_AA78E99F;
	{attribute addProperty Name "WcState"}
	WcState : WcState_98A4DF75;
	{attribute addProperty Name "InfoData"}
	InfoData : InfoData_0BDED7BF;
END_STRUCT
END_TYPE

// ---- DUTs/IO/Boxes/ATH2050_3A2EE8A7.TcDUT
{attribute addProperty BoxType "ATH2050-5501-0022"}
{attribute addProperty Id "FB_InputsAT %I*FB_Inputs_369FA10F000FB_OutputsAT %Q*FB_Outputs_734938A41620WcStateAT %I*WcState_98A4DF7520.250InfoDataAT %I*InfoData_7231B2DD80100"}
{attribute addProperty CRC "1927848659"}
{attribute addProperty SizeInBites "98"}
{attribute addProperty SizeInBytes "12.25"}
TYPE ATH2050_3A2EE8A7 :
STRUCT
	{attribute addProperty Name "FB_Inputs"}
	FB_Inputs : FB_Inputs_369FA10F;
	{attribute addProperty Name "FB_Outputs"}
	FB_Outputs : FB_Outputs_734938A4;
	{attribute addProperty Name "WcState"}
	WcState : WcState_98A4DF75;
	{attribute addProperty Name "InfoData"}
	InfoData : InfoData_7231B2DD;
END_STRUCT
END_TYPE

// ---- DUTs/IO/Boxes/ATH2040_948A301E.TcDUT
{attribute addProperty BoxType "ATH2040-5250-0022"}
{attribute addProperty Id "FB_InputsAT %I*FB_Inputs_16F33527000FB_OutputsAT %Q*FB_Outputs_734938A41620WcStateAT %I*WcState_98A4DF7520.250InfoDataAT %I*InfoData_7231B2DD80100"}
{attribute addProperty CRC "1885320120"}
{attribute addProperty SizeInBites "98"}
{attribute addProperty SizeInBytes "12.25"}
TYPE ATH2040_948A301E :
STRUCT
	{attribute addProperty Name "FB_Inputs"}
	FB_Inputs : FB_Inputs_16F33527;
	{attribute addProperty Name "FB_Outputs"}
	FB_Outputs : FB_Outputs_734938A4;
	{attribute addProperty Name "WcState"}
	WcState : WcState_98A4DF75;
	{attribute addProperty Name "InfoData"}
	InfoData : InfoData_7231B2DD;
END_STRUCT
END_TYPE

// ---- DUTs/IO/Boxes/ATH2040_BA5A9548.TcDUT
{attribute addProperty BoxType "ATH2040-0250-0022"}
{attribute addProperty Id "CC_InputsAT %I*CC_Inputs_9818D8D8256320CC_OutputsAT %Q*CC_Outputs_AA78E99F256320WcStateAT %I*WcState_98A4DF7520.250InfoDataAT %I*InfoData_0BDED7BF144180"}
{attribute addProperty CRC "3298337665"}
{attribute addProperty SizeInBites "658"}
{attribute addProperty SizeInBytes "82.25"}
TYPE ATH2040_BA5A9548 :
STRUCT
	{attribute addProperty Name "CC_Inputs"}
	CC_Inputs : CC_Inputs_9818D8D8;
	{attribute addProperty Name "CC_Outputs"}
	CC_Outputs : CC_Outputs_AA78E99F;
	{attribute addProperty Name "WcState"}
	WcState : WcState_98A4DF75;
	{attribute addProperty Name "InfoData"}
	InfoData : InfoData_0BDED7BF;
END_STRUCT
END_TYPE

// ---- DUTs/IO/Boxes/ATH2050_BA5A9548.TcDUT
{attribute addProperty BoxType "ATH2050-0500-0022"}
{attribute addProperty Id "CC_InputsAT %I*CC_Inputs_9818D8D8256320CC_OutputsAT %Q*CC_Outputs_AA78E99F256320WcStateAT %I*WcState_98A4DF7520.250InfoDataAT %I*InfoData_0BDED7BF144180"}
{attribute addProperty CRC "3298337665"}
{attribute addProperty SizeInBites "658"}
{attribute addProperty SizeInBytes "82.25"}
TYPE ATH2050_BA5A9548 :
STRUCT
	{attribute addProperty Name "CC_Inputs"}
	CC_Inputs : CC_Inputs_9818D8D8;
	{attribute addProperty Name "CC_Outputs"}
	CC_Outputs : CC_Outputs_AA78E99F;
	{attribute addProperty Name "WcState"}
	WcState : WcState_98A4DF75;
	{attribute addProperty Name "InfoData"}
	InfoData : InfoData_0BDED7BF;
END_STRUCT
END_TYPE

// ---- DUTs/IO/Boxes/ATH2000_89B1CED8.TcDUT
{attribute addProperty BoxType "ATH2000-5250-0022"}
{attribute addProperty Id "FB_InputsAT %I*FB_Inputs_1B840CA3000FB_OutputsAT %Q*FB_Outputs_734938A41620WcStateAT %I*WcState_98A4DF7520.250InfoDataAT %I*InfoData_7231B2DD80100"}
{attribute addProperty CRC "1035832528"}
{attribute addProperty SizeInBites "98"}
{attribute addProperty SizeInBytes "12.25"}
TYPE ATH2000_89B1CED8 :
STRUCT
	{attribute addProperty Name "FB_Inputs"}
	FB_Inputs : FB_Inputs_1B840CA3;
	{attribute addProperty Name "FB_Outputs"}
	FB_Outputs : FB_Outputs_734938A4;
	{attribute addProperty Name "WcState"}
	WcState : WcState_98A4DF75;
	{attribute addProperty Name "InfoData"}
	InfoData : InfoData_7231B2DD;
END_STRUCT
END_TYPE

// ---- DUTs/IO/Boxes/AX2000_4A6B0158.TcDUT
{attribute addProperty BoxType "AX2000-B110-0000"}
{attribute addProperty Id "InputsAT %I*Inputs_352C0ED16480OutputsAT %Q*Outputs_39B5897F4860WcStateAT %I*WcState_98A4DF7520.250InfoDataAT %I*InfoData_6C7DEEF988110"}
{attribute addProperty CRC "4027785059"}
{attribute addProperty SizeInBites "202"}
{attribute addProperty SizeInBytes "25.25"}
TYPE AX2000_4A6B0158 :
STRUCT
	{attribute addProperty Name "Inputs"}
	Inputs : Inputs_352C0ED1;
	{attribute addProperty Name "Outputs"}
	Outputs : Outputs_39B5897F;
	{attribute addProperty Name "WcState"}
	WcState : WcState_98A4DF75;
	{attribute addProperty Name "InfoData"}
	InfoData : InfoData_6C7DEEF9;
END_STRUCT
END_TYPE

// ---- DUTs/IO/Boxes/AX5191_3FB01CDA.TcDUT
{attribute addProperty BoxType "AX5191-0000-0212-0212"}
{attribute addProperty Id "AT_xAT %I*AT_x_15FCA3A680100MDTAT %Q*MDT_C2B17B7F4860WcStateAT %I*WcState_98A4DF7520.250InfoDataAT %I*InfoData_AEB17F4D152190"}
{attribute addProperty CRC "2773434183"}
{attribute addProperty SizeInBites "282"}
{attribute addProperty SizeInBytes "35.25"}
TYPE AX5191_3FB01CDA :
STRUCT
	{attribute addProperty Name "AT_x"}
	AT_x : AT_x_15FCA3A6;
	{attribute addProperty Name "MDT"}
	MDT : MDT_C2B17B7F;
	{attribute addProperty Name "WcState"}
	WcState : WcState_98A4DF75;
	{attribute addProperty Name "InfoData"}
	InfoData : InfoData_AEB17F4D;
END_STRUCT
END_TYPE

// ---- DUTs/IO/Boxes/AX5118_47F5CC47.TcDUT
{attribute addProperty BoxType "AX5118-0000-0011-0011"}
{attribute addProperty Id "AT_xAT %I*AT_x_029F01154860MDTAT %Q*MDT_47A878CF4860WcStateAT %I*WcState_98A4DF7520.250InfoDataAT %I*InfoData_AEB17F4D152190"}
{attribute addProperty CRC "245682833"}
{attribute addProperty SizeInBites "250"}
{attribute addProperty SizeInBytes "31.25"}
TYPE AX5118_47F5CC47 :
STRUCT
	{attribute addProperty Name "AT_x"}
	AT_x : AT_x_029F0115;
	{attribute addProperty Name "MDT"}
	MDT : MDT_47A878CF;
	{attribute addProperty Name "WcState"}
	WcState : WcState_98A4DF75;
	{attribute addProperty Name "InfoData"}
	InfoData : InfoData_AEB17F4D;
END_STRUCT
END_TYPE

// ---- DUTs/IO/Boxes/AX5125_47F5CC47.TcDUT
{attribute addProperty BoxType "AX5125-0000-0011-0011"}
{attribute addProperty Id "AT_xAT %I*AT_x_029F01154860MDTAT %Q*MDT_47A878CF4860WcStateAT %I*WcState_98A4DF7520.250InfoDataAT %I*InfoData_AEB17F4D152190"}
{attribute addProperty CRC "245682833"}
{attribute addProperty SizeInBites "250"}
{attribute addProperty SizeInBytes "31.25"}
TYPE AX5125_47F5CC47 :
STRUCT
	{attribute addProperty Name "AT_x"}
	AT_x : AT_x_029F0115;
	{attribute addProperty Name "MDT"}
	MDT : MDT_47A878CF;
	{attribute addProperty Name "WcState"}
	WcState : WcState_98A4DF75;
	{attribute addProperty Name "InfoData"}
	InfoData : InfoData_AEB17F4D;
END_STRUCT
END_TYPE

// ---- DUTs/IO/Boxes/AX5201_D0280DF2.TcDUT
{attribute addProperty BoxType "AX5201-0000-0011-0011"}
{attribute addProperty Id "AT_xAT %I*ARRAY[0..2] OF AT_029F011596120MDTAT %Q*ARRAY[0..2] OF MDT_47A878CF96120WcStateAT %I*WcState_98A4DF7520.250InfoDataAT %I*InfoData_81099714160200"}
{attribute addProperty CRC "1275577876"}
{attribute addProperty SizeInBites "354"}
{attribute addProperty SizeInBytes "44.25"}
TYPE AX5201_D0280DF2 :
STRUCT
	{attribute addProperty Name "AT"}
	AT_x : ARRAY[0..2] OF AT_029F0115;
	{attribute addProperty Name "MDT"}
	MDT : ARRAY[0..2] OF MDT_47A878CF;
	{attribute addProperty Name "WcState"}
	WcState : WcState_98A4DF75;
	{attribute addProperty Name "InfoData"}
	InfoData : InfoData_81099714;
END_STRUCT
END_TYPE

// ---- DUTs/IO/Boxes/AX5106_47F5CC47.TcDUT
{attribute addProperty BoxType "AX5106-0000-0010-0010"}
{attribute addProperty Id "AT_xAT %I*AT_x_029F01154860MDTAT %Q*MDT_47A878CF4860WcStateAT %I*WcState_98A4DF7520.250InfoDataAT %I*InfoData_AEB17F4D152190"}
{attribute addProperty CRC "245682833"}
{attribute addProperty SizeInBites "250"}
{attribute addProperty SizeInBytes "31.25"}
TYPE AX5106_47F5CC47 :
STRUCT
	{attribute addProperty Name "AT_x"}
	AT_x : AT_x_029F0115;
	{attribute addProperty Name "MDT"}
	MDT : MDT_47A878CF;
	{attribute addProperty Name "WcState"}
	WcState : WcState_98A4DF75;
	{attribute addProperty Name "InfoData"}
	InfoData : InfoData_AEB17F4D;
END_STRUCT
END_TYPE

// ---- DUTs/IO/Boxes/AX5112_47F5CC47.TcDUT
{attribute addProperty BoxType "AX5112-0000-0010-0010"}
{attribute addProperty Id "AT_xAT %I*AT_x_029F01154860MDTAT %Q*MDT_47A878CF4860WcStateAT %I*WcState_98A4DF7520.250InfoDataAT %I*InfoData_AEB17F4D152190"}
{attribute addProperty CRC "245682833"}
{attribute addProperty SizeInBites "250"}
{attribute addProperty SizeInBytes "31.25"}
TYPE AX5112_47F5CC47 :
STRUCT
	{attribute addProperty Name "AT_x"}
	AT_x : AT_x_029F0115;
	{attribute addProperty Name "MDT"}
	MDT : MDT_47A878CF;
	{attribute addProperty Name "WcState"}
	WcState : WcState_98A4DF75;
	{attribute addProperty Name "InfoData"}
	InfoData : InfoData_AEB17F4D;
END_STRUCT
END_TYPE

// ---- DUTs/IO/Boxes/AX5103_47F5CC47.TcDUT
{attribute addProperty BoxType "AX5103-0000-0007-0007"}
{attribute addProperty Id "AT_xAT %I*AT_x_029F01154860MDTAT %Q*MDT_47A878CF4860WcStateAT %I*WcState_98A4DF7520.250InfoDataAT %I*InfoData_AEB17F4D152190"}
{attribute addProperty CRC "245682833"}
{attribute addProperty SizeInBites "250"}
{attribute addProperty SizeInBytes "31.25"}
TYPE AX5103_47F5CC47 :
STRUCT
	{attribute addProperty Name "AT_x"}
	AT_x : AT_x_029F0115;
	{attribute addProperty Name "MDT"}
	MDT : MDT_47A878CF;
	{attribute addProperty Name "WcState"}
	WcState : WcState_98A4DF75;
	{attribute addProperty Name "InfoData"}
	InfoData : InfoData_AEB17F4D;
END_STRUCT
END_TYPE

// ---- DUTs/IO/Boxes/AX5101_47F5CC47.TcDUT
{attribute addProperty BoxType "AX5101-0000-0005-0005"}
{attribute addProperty Id "AT_xAT %I*AT_x_029F01154860MDTAT %Q*MDT_47A878CF4860WcStateAT %I*WcState_98A4DF7520.250InfoDataAT %I*InfoData_AEB17F4D152190"}
{attribute addProperty CRC "245682833"}
{attribute addProperty SizeInBites "250"}
{attribute addProperty SizeInBytes "31.25"}
TYPE AX5101_47F5CC47 :
STRUCT
	{attribute addProperty Name "AT_x"}
	AT_x : AT_x_029F0115;
	{attribute addProperty Name "MDT"}
	MDT : MDT_47A878CF;
	{attribute addProperty Name "WcState"}
	WcState : WcState_98A4DF75;
	{attribute addProperty Name "InfoData"}
	InfoData : InfoData_AEB17F4D;
END_STRUCT
END_TYPE

// ---- DUTs/IO/Boxes/AX5203_D0280DF2.TcDUT
{attribute addProperty BoxType "AX5203-0000-0005-0005"}
{attribute addProperty Id "AT_xAT %I*ARRAY[0..2] OF AT_029F011596120MDTAT %Q*ARRAY[0..2] OF MDT_47A878CF96120WcStateAT %I*WcState_98A4DF7520.250InfoDataAT %I*InfoData_81099714160200"}
{attribute addProperty CRC "1275577876"}
{attribute addProperty SizeInBites "354"}
{attribute addProperty SizeInBytes "44.25"}
TYPE AX5203_D0280DF2 :
STRUCT
	{attribute addProperty Name "AT"}
	AT_x : ARRAY[0..2] OF AT_029F0115;
	{attribute addProperty Name "MDT"}
	MDT : ARRAY[0..2] OF MDT_47A878CF;
	{attribute addProperty Name "WcState"}
	WcState : WcState_98A4DF75;
	{attribute addProperty Name "InfoData"}
	InfoData : InfoData_81099714;
END_STRUCT
END_TYPE

// ---- DUTs/IO/Boxes/AX5206_D0280DF2.TcDUT
{attribute addProperty BoxType "AX5206-0000-0005-0005"}
{attribute addProperty Id "AT_xAT %I*ARRAY[0..2] OF AT_029F011596120MDTAT %Q*ARRAY[0..2] OF MDT_47A878CF96120WcStateAT %I*WcState_98A4DF7520.250InfoDataAT %I*InfoData_81099714160200"}
{attribute addProperty CRC "1275577876"}
{attribute addProperty SizeInBites "354"}
{attribute addProperty SizeInBytes "44.25"}
TYPE AX5206_D0280DF2 :
STRUCT
	{attribute addProperty Name "AT"}
	AT_x : ARRAY[0..2] OF AT_029F0115;
	{attribute addProperty Name "MDT"}
	MDT : ARRAY[0..2] OF MDT_47A878CF;
	{attribute addProperty Name "WcState"}
	WcState : WcState_98A4DF75;
	{attribute addProperty Name "InfoData"}
	InfoData : InfoData_81099714;
END_STRUCT
END_TYPE

// ---- DUTs/IO/Boxes/AX5021_292ACD47.TcDUT
{attribute addProperty BoxType "AX5021-0000-0002-0002"}
{attribute addProperty Id "AT_xAT %I*AT_x_F64797681620MDTAT %Q*MDT_81E4A3441620WcStateAT %I*WcState_98A4DF7520.250InfoDataAT %I*InfoData_AEB17F4D152190"}
{attribute addProperty CRC "2967045990"}
{attribute addProperty SizeInBites "186"}
{attribute addProperty SizeInBytes "23.25"}
TYPE AX5021_292ACD47 :
STRUCT
	{attribute addProperty Name "AT_x"}
	AT_x : AT_x_F6479768;
	{attribute addProperty Name "MDT"}
	MDT : MDT_81E4A344;
	{attribute addProperty Name "WcState"}
	WcState : WcState_98A4DF75;
	{attribute addProperty Name "InfoData"}
	InfoData : InfoData_AEB17F4D;
END_STRUCT
END_TYPE

// ---- DUTs/IO/Boxes/AX5206_7BA23180.TcDUT
{attribute addProperty BoxType "AX5206-0000-0200-0200"}
{attribute addProperty Id "AT_xAT %I*ARRAY[0..3] OF AT_15FCA3A6160200MDTAT %Q*ARRAY[0..2] OF MDT_C2B17B7F96120WcStateAT %I*WcState_98A4DF7520.250InfoDataAT %I*InfoData_81099714160200"}
{attribute addProperty CRC "2852748137"}
{attribute addProperty SizeInBites "418"}
{attribute addProperty SizeInBytes "52.25"}
TYPE AX5206_7BA23180 :
STRUCT
	{attribute addProperty Name "AT"}
	AT_x : ARRAY[0..3] OF AT_15FCA3A6;
	{attribute addProperty Name "MDT"}
	MDT : ARRAY[0..2] OF MDT_C2B17B7F;
	{attribute addProperty Name "WcState"}
	WcState : WcState_98A4DF75;
	{attribute addProperty Name "InfoData"}
	InfoData : InfoData_81099714;
END_STRUCT
END_TYPE

// ---- DUTs/IO/Boxes/AX5140_3FB01CDA.TcDUT
{attribute addProperty BoxType "AX5140-0000-0200-0200"}
{attribute addProperty Id "AT_xAT %I*AT_x_15FCA3A680100MDTAT %Q*MDT_C2B17B7F4860WcStateAT %I*WcState_98A4DF7520.250InfoDataAT %I*InfoData_AEB17F4D152190"}
{attribute addProperty CRC "2773434183"}
{attribute addProperty SizeInBites "282"}
{attribute addProperty SizeInBytes "35.25"}
TYPE AX5140_3FB01CDA :
STRUCT
	{attribute addProperty Name "AT_x"}
	AT_x : AT_x_15FCA3A6;
	{attribute addProperty Name "MDT"}
	MDT : MDT_C2B17B7F;
	{attribute addProperty Name "WcState"}
	WcState : WcState_98A4DF75;
	{attribute addProperty Name "InfoData"}
	InfoData : InfoData_AEB17F4D;
END_STRUCT
END_TYPE

// ---- DUTs/IO/Boxes/AX5118_3FB01CDA.TcDUT
{attribute addProperty BoxType "AX5118-0000-0200-0200"}
{attribute addProperty Id "AT_xAT %I*AT_x_15FCA3A680100MDTAT %Q*MDT_C2B17B7F4860WcStateAT %I*WcState_98A4DF7520.250InfoDataAT %I*InfoData_AEB17F4D152190"}
{attribute addProperty CRC "2773434183"}
{attribute addProperty SizeInBites "282"}
{attribute addProperty SizeInBytes "35.25"}
TYPE AX5118_3FB01CDA :
STRUCT
	{attribute addProperty Name "AT_x"}
	AT_x : AT_x_15FCA3A6;
	{attribute addProperty Name "MDT"}
	MDT : MDT_C2B17B7F;
	{attribute addProperty Name "WcState"}
	WcState : WcState_98A4DF75;
	{attribute addProperty Name "InfoData"}
	InfoData : InfoData_AEB17F4D;
END_STRUCT
END_TYPE

// ---- DUTs/IO/Boxes/AX5125_3FB01CDA.TcDUT
{attribute addProperty BoxType "AX5125-0000-0201-0201"}
{attribute addProperty Id "AT_xAT %I*AT_x_15FCA3A680100MDTAT %Q*MDT_C2B17B7F4860WcStateAT %I*WcState_98A4DF7520.250InfoDataAT %I*InfoData_AEB17F4D152190"}
{attribute addProperty CRC "2773434183"}
{attribute addProperty SizeInBites "282"}
{attribute addProperty SizeInBytes "35.25"}
TYPE AX5125_3FB01CDA :
STRUCT
	{attribute addProperty Name "AT_x"}
	AT_x : AT_x_15FCA3A6;
	{attribute addProperty Name "MDT"}
	MDT : MDT_C2B17B7F;
	{attribute addProperty Name "WcState"}
	WcState : WcState_98A4DF75;
	{attribute addProperty Name "InfoData"}
	InfoData : InfoData_AEB17F4D;
END_STRUCT
END_TYPE

// ---- DUTs/IO/Boxes/AX5101_3FB01CDA.TcDUT
{attribute addProperty BoxType "AX5101-0000-0202-0202"}
{attribute addProperty Id "AT_xAT %I*AT_x_15FCA3A680100MDTAT %Q*MDT_C2B17B7F4860WcStateAT %I*WcState_98A4DF7520.250InfoDataAT %I*InfoData_AEB17F4D152190"}
{attribute addProperty CRC "2773434183"}
{attribute addProperty SizeInBites "282"}
{attribute addProperty SizeInBytes "35.25"}
TYPE AX5101_3FB01CDA :
STRUCT
	{attribute addProperty Name "AT_x"}
	AT_x : AT_x_15FCA3A6;
	{attribute addProperty Name "MDT"}
	MDT : MDT_C2B17B7F;
	{attribute addProperty Name "WcState"}
	WcState : WcState_98A4DF75;
	{attribute addProperty Name "InfoData"}
	InfoData : InfoData_AEB17F4D;
END_STRUCT
END_TYPE

// ---- DUTs/IO/Boxes/AX5172_3FB01CDA.TcDUT
{attribute addProperty BoxType "AX5172-0000-0203-0203"}
{attribute addProperty Id "AT_xAT %I*AT_x_15FCA3A680100MDTAT %Q*MDT_C2B17B7F4860WcStateAT %I*WcState_98A4DF7520.250InfoDataAT %I*InfoData_AEB17F4D152190"}
{attribute addProperty CRC "2773434183"}
{attribute addProperty SizeInBites "282"}
{attribute addProperty SizeInBytes "35.25"}
TYPE AX5172_3FB01CDA :
STRUCT
	{attribute addProperty Name "AT_x"}
	AT_x : AT_x_15FCA3A6;
	{attribute addProperty Name "MDT"}
	MDT : MDT_C2B17B7F;
	{attribute addProperty Name "WcState"}
	WcState : WcState_98A4DF75;
	{attribute addProperty Name "InfoData"}
	InfoData : InfoData_AEB17F4D;
END_STRUCT
END_TYPE

// ---- DUTs/IO/Boxes/AX5106_3FB01CDA.TcDUT
{attribute addProperty BoxType "AX5106-0000-0203-0203"}
{attribute addProperty Id "AT_xAT %I*AT_x_15FCA3A680100MDTAT %Q*MDT_C2B17B7F4860WcStateAT %I*WcState_98A4DF7520.250InfoDataAT %I*InfoData_AEB17F4D152190"}
{attribute addProperty CRC "2773434183"}
{attribute addProperty SizeInBites "282"}
{attribute addProperty SizeInBytes "35.25"}
TYPE AX5106_3FB01CDA :
STRUCT
	{attribute addProperty Name "AT_x"}
	AT_x : AT_x_15FCA3A6;
	{attribute addProperty Name "MDT"}
	MDT : MDT_C2B17B7F;
	{attribute addProperty Name "WcState"}
	WcState : WcState_98A4DF75;
	{attribute addProperty Name "InfoData"}
	InfoData : InfoData_AEB17F4D;
END_STRUCT
END_TYPE

// ---- DUTs/IO/Boxes/AX5203_7BA23180.TcDUT
{attribute addProperty BoxType "AX5203-0000-0210-0210"}
{attribute addProperty Id "AT_xAT %I*ARRAY[0..3] OF AT_15FCA3A6160200MDTAT %Q*ARRAY[0..2] OF MDT_C2B17B7F96120WcStateAT %I*WcState_98A4DF7520.250InfoDataAT %I*InfoData_81099714160200"}
{attribute addProperty CRC "2852748137"}
{attribute addProperty SizeInBites "418"}
{attribute addProperty SizeInBytes "52.25"}
TYPE AX5203_7BA23180 :
STRUCT
	{attribute addProperty Name "AT"}
	AT_x : ARRAY[0..3] OF AT_15FCA3A6;
	{attribute addProperty Name "MDT"}
	MDT : ARRAY[0..2] OF MDT_C2B17B7F;
	{attribute addProperty Name "WcState"}
	WcState : WcState_98A4DF75;
	{attribute addProperty Name "InfoData"}
	InfoData : InfoData_81099714;
END_STRUCT
END_TYPE

// ---- DUTs/IO/Boxes/AX5193_3FB01CDA.TcDUT
{attribute addProperty BoxType "AX5193-0000-0210-0210"}
{attribute addProperty Id "AT_xAT %I*AT_x_15FCA3A680100MDTAT %Q*MDT_C2B17B7F4860WcStateAT %I*WcState_98A4DF7520.250InfoDataAT %I*InfoData_AEB17F4D152190"}
{attribute addProperty CRC "2773434183"}
{attribute addProperty SizeInBites "282"}
{attribute addProperty SizeInBytes "35.25"}
TYPE AX5193_3FB01CDA :
STRUCT
	{attribute addProperty Name "AT_x"}
	AT_x : AT_x_15FCA3A6;
	{attribute addProperty Name "MDT"}
	MDT : MDT_C2B17B7F;
	{attribute addProperty Name "WcState"}
	WcState : WcState_98A4DF75;
	{attribute addProperty Name "InfoData"}
	InfoData : InfoData_AEB17F4D;
END_STRUCT
END_TYPE

// ---- DUTs/IO/Boxes/AX5192_3FB01CDA.TcDUT
{attribute addProperty BoxType "AX5192-0000-0210-0210"}
{attribute addProperty Id "AT_xAT %I*AT_x_15FCA3A680100MDTAT %Q*MDT_C2B17B7F4860WcStateAT %I*WcState_98A4DF7520.250InfoDataAT %I*InfoData_AEB17F4D152190"}
{attribute addProperty CRC "2773434183"}
{attribute addProperty SizeInBites "282"}
{attribute addProperty SizeInBytes "35.25"}
TYPE AX5192_3FB01CDA :
STRUCT
	{attribute addProperty Name "AT_x"}
	AT_x : AT_x_15FCA3A6;
	{attribute addProperty Name "MDT"}
	MDT : MDT_C2B17B7F;
	{attribute addProperty Name "WcState"}
	WcState : WcState_98A4DF75;
	{attribute addProperty Name "InfoData"}
	InfoData : InfoData_AEB17F4D;
END_STRUCT
END_TYPE

// ---- DUTs/IO/Boxes/AX5160_3FB01CDA.TcDUT
{attribute addProperty BoxType "AX5160-0000-0210-0210"}
{attribute addProperty Id "AT_xAT %I*AT_x_15FCA3A680100MDTAT %Q*MDT_C2B17B7F4860WcStateAT %I*WcState_98A4DF7520.250InfoDataAT %I*InfoData_AEB17F4D152190"}
{attribute addProperty CRC "2773434183"}
{attribute addProperty SizeInBites "282"}
{attribute addProperty SizeInBytes "35.25"}
TYPE AX5160_3FB01CDA :
STRUCT
	{attribute addProperty Name "AT_x"}
	AT_x : AT_x_15FCA3A6;
	{attribute addProperty Name "MDT"}
	MDT : MDT_C2B17B7F;
	{attribute addProperty Name "WcState"}
	WcState : WcState_98A4DF75;
	{attribute addProperty Name "InfoData"}
	InfoData : InfoData_AEB17F4D;
END_STRUCT
END_TYPE

// ---- DUTs/IO/Boxes/AX5112_3FB01CDA.TcDUT
{attribute addProperty BoxType "AX5112-0000-0210-0210"}
{attribute addProperty Id "AT_xAT %I*AT_x_15FCA3A680100MDTAT %Q*MDT_C2B17B7F4860WcStateAT %I*WcState_98A4DF7520.250InfoDataAT %I*InfoData_AEB17F4D152190"}
{attribute addProperty CRC "2773434183"}
{attribute addProperty SizeInBites "282"}
{attribute addProperty SizeInBytes "35.25"}
TYPE AX5112_3FB01CDA :
STRUCT
	{attribute addProperty Name "AT_x"}
	AT_x : AT_x_15FCA3A6;
	{attribute addProperty Name "MDT"}
	MDT : MDT_C2B17B7F;
	{attribute addProperty Name "WcState"}
	WcState : WcState_98A4DF75;
	{attribute addProperty Name "InfoData"}
	InfoData : InfoData_AEB17F4D;
END_STRUCT
END_TYPE

// ---- DUTs/IO/Boxes/AX5201_7BA23180.TcDUT
{attribute addProperty BoxType "AX5201-0000-0200-0200"}
{attribute addProperty Id "AT_xAT %I*ARRAY[0..3] OF AT_15FCA3A6160200MDTAT %Q*ARRAY[0..2] OF MDT_C2B17B7F96120WcStateAT %I*WcState_98A4DF7520.250InfoDataAT %I*InfoData_81099714160200"}
{attribute addProperty CRC "2852748137"}
{attribute addProperty SizeInBites "418"}
{attribute addProperty SizeInBytes "52.25"}
TYPE AX5201_7BA23180 :
STRUCT
	{attribute addProperty Name "AT"}
	AT_x : ARRAY[0..3] OF AT_15FCA3A6;
	{attribute addProperty Name "MDT"}
	MDT : ARRAY[0..2] OF MDT_C2B17B7F;
	{attribute addProperty Name "WcState"}
	WcState : WcState_98A4DF75;
	{attribute addProperty Name "InfoData"}
	InfoData : InfoData_81099714;
END_STRUCT
END_TYPE

// ---- DUTs/IO/Boxes/AX5103_3FB01CDA.TcDUT
{attribute addProperty BoxType "AX5103-0000-0201-0201"}
{attribute addProperty Id "AT_xAT %I*AT_x_15FCA3A680100MDTAT %Q*MDT_C2B17B7F4860WcStateAT %I*WcState_98A4DF7520.250InfoDataAT %I*InfoData_AEB17F4D152190"}
{attribute addProperty CRC "2773434183"}
{attribute addProperty SizeInBites "282"}
{attribute addProperty SizeInBytes "35.25"}
TYPE AX5103_3FB01CDA :
STRUCT
	{attribute addProperty Name "AT_x"}
	AT_x : AT_x_15FCA3A6;
	{attribute addProperty Name "MDT"}
	MDT : MDT_C2B17B7F;
	{attribute addProperty Name "WcState"}
	WcState : WcState_98A4DF75;
	{attribute addProperty Name "InfoData"}
	InfoData : InfoData_AEB17F4D;
END_STRUCT
END_TYPE

// ---- DUTs/IO/Boxes/AX5190_3FB01CDA.TcDUT
{attribute addProperty BoxType "AX5190-0000-0203-0203"}
{attribute addProperty Id "AT_xAT %I*AT_x_15FCA3A680100MDTAT %Q*MDT_C2B17B7F4860WcStateAT %I*WcState_98A4DF7520.250InfoDataAT %I*InfoData_AEB17F4D152190"}
{attribute addProperty CRC "2773434183"}
{attribute addProperty SizeInBites "282"}
{attribute addProperty SizeInBytes "35.25"}
TYPE AX5190_3FB01CDA :
STRUCT
	{attribute addProperty Name "AT_x"}
	AT_x : AT_x_15FCA3A6;
	{attribute addProperty Name "MDT"}
	MDT : MDT_C2B17B7F;
	{attribute addProperty Name "WcState"}
	WcState : WcState_98A4DF75;
	{attribute addProperty Name "InfoData"}
	InfoData : InfoData_AEB17F4D;
END_STRUCT
END_TYPE

// ---- DUTs/IO/Boxes/AMP8000_2B905711.TcDUT
{attribute addProperty BoxType "AMP8000-0000-0103-0103"}
{attribute addProperty Id "DeviceDevice_F82A60211620Ch_ACh_A_B17182A2176220WcStateAT %I*WcState_98A4DF7520.250InfoDataAT %I*InfoData_F030DC9B200250"}
{attribute addProperty CRC "3898025815"}
{attribute addProperty SizeInBites "394"}
{attribute addProperty SizeInBytes "49.25"}
TYPE AMP8000_2B905711 :
STRUCT
	{attribute addProperty Name "Device"}
	Device : Device_F82A6021;
	{attribute addProperty Name "Ch_A"}
	Ch_A : Ch_A_B17182A2;
	{attribute addProperty Name "WcState"}
	WcState : WcState_98A4DF75;
	{attribute addProperty Name "InfoData"}
	InfoData : InfoData_F030DC9B;
END_STRUCT
END_TYPE

// ---- DUTs/IO/Boxes/AMP8000_5E0E86F8.TcDUT
{attribute addProperty BoxType "AMP8000-0030-0103-0103"}
{attribute addProperty Id "DeviceDevice_F82A60211620Device_SafetyDevice_Safety_AF71BE9D160200Ch_ACh_A_B17182A2176220WcStateAT %I*WcState_DC9C971540.50InfoDataAT %I*InfoData_F030DC9B200250"}
{attribute addProperty CRC "4031425745"}
{attribute addProperty SizeInBites "556"}
{attribute addProperty SizeInBytes "69.5"}
TYPE AMP8000_5E0E86F8 :
STRUCT
	{attribute addProperty Name "Device"}
	Device : Device_F82A6021;
	{attribute addProperty Name "Device_Safety"}
	Device_Safety : Device_Safety_AF71BE9D;
	{attribute addProperty Name "Ch_A"}
	Ch_A : Ch_A_B17182A2;
	{attribute addProperty Name "WcState"}
	WcState : WcState_DC9C9715;
	{attribute addProperty Name "InfoData"}
	InfoData : InfoData_F030DC9B;
END_STRUCT
END_TYPE

// ---- DUTs/IO/Boxes/AX8108_E3898C73.TcDUT
{attribute addProperty BoxType "AX8108-0000-0041-0041"}
{attribute addProperty Id "DeviceDevice_FD48B4B01620Ch_ACh_A_99F8614F240300WcStateAT %I*WcState_98A4DF7520.250InfoDataAT %I*InfoData_F030DC9B200250"}
{attribute addProperty CRC "1708484915"}
{attribute addProperty SizeInBites "458"}
{attribute addProperty SizeInBytes "57.25"}
TYPE AX8108_E3898C73 :
STRUCT
	{attribute addProperty Name "Device"}
	Device : Device_FD48B4B0;
	{attribute addProperty Name "Ch_A"}
	Ch_A : Ch_A_99F8614F;
	{attribute addProperty Name "WcState"}
	WcState : WcState_98A4DF75;
	{attribute addProperty Name "InfoData"}
	InfoData : InfoData_F030DC9B;
END_STRUCT
END_TYPE

// ---- DUTs/IO/Boxes/AX8108_6822C7B9.TcDUT
{attribute addProperty BoxType "AX8108-0000-0100-0100"}
{attribute addProperty Id "DeviceDevice_F82A60211620Ch_ACh_A_359CD49A176220WcStateAT %I*WcState_98A4DF7520.250InfoDataAT %I*InfoData_F030DC9B200250"}
{attribute addProperty CRC "2011418308"}
{attribute addProperty SizeInBites "394"}
{attribute addProperty SizeInBytes "49.25"}
TYPE AX8108_6822C7B9 :
STRUCT
	{attribute addProperty Name "Device"}
	Device : Device_F82A6021;
	{attribute addProperty Name "Ch_A"}
	Ch_A : Ch_A_359CD49A;
	{attribute addProperty Name "WcState"}
	WcState : WcState_98A4DF75;
	{attribute addProperty Name "InfoData"}
	InfoData : InfoData_F030DC9B;
END_STRUCT
END_TYPE

// ---- DUTs/IO/Boxes/AX8108_2B905711.TcDUT
{attribute addProperty BoxType "AX8108-0000-0102-0102"}
{attribute addProperty Id "DeviceDevice_F82A60211620Ch_ACh_A_B17182A2176220WcStateAT %I*WcState_98A4DF7520.250InfoDataAT %I*InfoData_F030DC9B200250"}
{attribute addProperty CRC "3898025815"}
{attribute addProperty SizeInBites "394"}
{attribute addProperty SizeInBytes "49.25"}
TYPE AX8108_2B905711 :
STRUCT
	{attribute addProperty Name "Device"}
	Device : Device_F82A6021;
	{attribute addProperty Name "Ch_A"}
	Ch_A : Ch_A_B17182A2;
	{attribute addProperty Name "WcState"}
	WcState : WcState_98A4DF75;
	{attribute addProperty Name "InfoData"}
	InfoData : InfoData_F030DC9B;
END_STRUCT
END_TYPE

// ---- DUTs/IO/Boxes/AX8108_E4DF8033.TcDUT
{attribute addProperty BoxType "AX8108-0100-0101-0101"}
{attribute addProperty Id "DeviceDevice_F82A60211620Device_SafetyDevice_Safety_AF71BE9D160200Ch_ACh_A_359CD49A176220WcStateAT %I*WcState_DC9C971540.50InfoDataAT %I*InfoData_F030DC9B200250"}
{attribute addProperty CRC "1051991048"}
{attribute addProperty SizeInBites "556"}
{attribute addProperty SizeInBytes "69.5"}
TYPE AX8108_E4DF8033 :
STRUCT
	{attribute addProperty Name "Device"}
	Device : Device_F82A6021;
	{attribute addProperty Name "Device_Safety"}
	Device_Safety : Device_Safety_AF71BE9D;
	{attribute addProperty Name "Ch_A"}
	Ch_A : Ch_A_359CD49A;
	{attribute addProperty Name "WcState"}
	WcState : WcState_DC9C9715;
	{attribute addProperty Name "InfoData"}
	InfoData : InfoData_F030DC9B;
END_STRUCT
END_TYPE

// ---- DUTs/IO/Boxes/AX8108_5E0E86F8.TcDUT
{attribute addProperty BoxType "AX8108-0100-0102-0102"}
{attribute addProperty Id "DeviceDevice_F82A60211620Device_SafetyDevice_Safety_AF71BE9D160200Ch_ACh_A_B17182A2176220WcStateAT %I*WcState_DC9C971540.50InfoDataAT %I*InfoData_F030DC9B200250"}
{attribute addProperty CRC "4031425745"}
{attribute addProperty SizeInBites "556"}
{attribute addProperty SizeInBytes "69.5"}
TYPE AX8108_5E0E86F8 :
STRUCT
	{attribute addProperty Name "Device"}
	Device : Device_F82A6021;
	{attribute addProperty Name "Device_Safety"}
	Device_Safety : Device_Safety_AF71BE9D;
	{attribute addProperty Name "Ch_A"}
	Ch_A : Ch_A_B17182A2;
	{attribute addProperty Name "WcState"}
	WcState : WcState_DC9C9715;
	{attribute addProperty Name "InfoData"}
	InfoData : InfoData_F030DC9B;
END_STRUCT
END_TYPE

// ---- DUTs/IO/Boxes/AX8118_E3898C73.TcDUT
{attribute addProperty BoxType "AX8118-0000-0041-0041"}
{attribute addProperty Id "DeviceDevice_FD48B4B01620Ch_ACh_A_99F8614F240300WcStateAT %I*WcState_98A4DF7520.250InfoDataAT %I*InfoData_F030DC9B200250"}
{attribute addProperty CRC "1708484915"}
{attribute addProperty SizeInBites "458"}
{attribute addProperty SizeInBytes "57.25"}
TYPE AX8118_E3898C73 :
STRUCT
	{attribute addProperty Name "Device"}
	Device : Device_FD48B4B0;
	{attribute addProperty Name "Ch_A"}
	Ch_A : Ch_A_99F8614F;
	{attribute addProperty Name "WcState"}
	WcState : WcState_98A4DF75;
	{attribute addProperty Name "InfoData"}
	InfoData : InfoData_F030DC9B;
END_STRUCT
END_TYPE

// ---- DUTs/IO/Boxes/AX8118_6822C7B9.TcDUT
{attribute addProperty BoxType "AX8118-0000-0100-0100"}
{attribute addProperty Id "DeviceDevice_F82A60211620Ch_ACh_A_359CD49A176220WcStateAT %I*WcState_98A4DF7520.250InfoDataAT %I*InfoData_F030DC9B200250"}
{attribute addProperty CRC "2011418308"}
{attribute addProperty SizeInBites "394"}
{attribute addProperty SizeInBytes "49.25"}
TYPE AX8118_6822C7B9 :
STRUCT
	{attribute addProperty Name "Device"}
	Device : Device_F82A6021;
	{attribute addProperty Name "Ch_A"}
	Ch_A : Ch_A_359CD49A;
	{attribute addProperty Name "WcState"}
	WcState : WcState_98A4DF75;
	{attribute addProperty Name "InfoData"}
	InfoData : InfoData_F030DC9B;
END_STRUCT
END_TYPE

// ---- DUTs/IO/Boxes/AX8118_2B905711.TcDUT
{attribute addProperty BoxType "AX8118-0000-0102-0102"}
{attribute addProperty Id "DeviceDevice_F82A60211620Ch_ACh_A_B17182A2176220WcStateAT %I*WcState_98A4DF7520.250InfoDataAT %I*InfoData_F030DC9B200250"}
{attribute addProperty CRC "3898025815"}
{attribute addProperty SizeInBites "394"}
{attribute addProperty SizeInBytes "49.25"}
TYPE AX8118_2B905711 :
STRUCT
	{attribute addProperty Name "Device"}
	Device : Device_F82A6021;
	{attribute addProperty Name "Ch_A"}
	Ch_A : Ch_A_B17182A2;
	{attribute addProperty Name "WcState"}
	WcState : WcState_98A4DF75;
	{attribute addProperty Name "InfoData"}
	InfoData : InfoData_F030DC9B;
END_STRUCT
END_TYPE

// ---- DUTs/IO/Boxes/AX8118_E4DF8033.TcDUT
{attribute addProperty BoxType "AX8118-0100-0101-0101"}
{attribute addProperty Id "DeviceDevice_F82A60211620Device_SafetyDevice_Safety_AF71BE9D160200Ch_ACh_A_359CD49A176220WcStateAT %I*WcState_DC9C971540.50InfoDataAT %I*InfoData_F030DC9B200250"}
{attribute addProperty CRC "1051991048"}
{attribute addProperty SizeInBites "556"}
{attribute addProperty SizeInBytes "69.5"}
TYPE AX8118_E4DF8033 :
STRUCT
	{attribute addProperty Name "Device"}
	Device : Device_F82A6021;
	{attribute addProperty Name "Device_Safety"}
	Device_Safety : Device_Safety_AF71BE9D;
	{attribute addProperty Name "Ch_A"}
	Ch_A : Ch_A_359CD49A;
	{attribute addProperty Name "WcState"}
	WcState : WcState_DC9C9715;
	{attribute addProperty Name "InfoData"}
	InfoData : InfoData_F030DC9B;
END_STRUCT
END_TYPE

// ---- DUTs/IO/Boxes/AX8118_5E0E86F8.TcDUT
{attribute addProperty BoxType "AX8118-0100-0102-0102"}
{attribute addProperty Id "DeviceDevice_F82A60211620Device_SafetyDevice_Safety_AF71BE9D160200Ch_ACh_A_B17182A2176220WcStateAT %I*WcState_DC9C971540.50InfoDataAT %I*InfoData_F030DC9B200250"}
{attribute addProperty CRC "4031425745"}
{attribute addProperty SizeInBites "556"}
{attribute addProperty SizeInBytes "69.5"}
TYPE AX8118_5E0E86F8 :
STRUCT
	{attribute addProperty Name "Device"}
	Device : Device_F82A6021;
	{attribute addProperty Name "Device_Safety"}
	Device_Safety : Device_Safety_AF71BE9D;
	{attribute addProperty Name "Ch_A"}
	Ch_A : Ch_A_B17182A2;
	{attribute addProperty Name "WcState"}
	WcState : WcState_DC9C9715;
	{attribute addProperty Name "InfoData"}
	InfoData : InfoData_F030DC9B;
END_STRUCT
END_TYPE

// ---- DUTs/IO/Boxes/AX8206_C98B9CD1.TcDUT
{attribute addProperty BoxType "AX8206-0000-0041-0041"}
{attribute addProperty Id "DeviceDevice_FD48B4B01620Ch_ACh_A_99F8614F240300Ch_BCh_B_5DC205AF240300WcStateAT %I*WcState_98A4DF7520.250InfoDataAT %I*InfoData_17277C5A208260"}
{attribute addProperty CRC "1253737747"}
{attribute addProperty SizeInBites "706"}
{attribute addProperty SizeInBytes "88.25"}
TYPE AX8206_C98B9CD1 :
STRUCT
	{attribute addProperty Name "Device"}
	Device : Device_FD48B4B0;
	{attribute addProperty Name "Ch_A"}
	Ch_A : Ch_A_99F8614F;
	{attribute addProperty Name "Ch_B"}
	Ch_B : Ch_B_5DC205AF;
	{attribute addProperty Name "WcState"}
	WcState : WcState_98A4DF75;
	{attribute addProperty Name "InfoData"}
	InfoData : InfoData_17277C5A;
END_STRUCT
END_TYPE

// ---- DUTs/IO/Boxes/AX8206_06F284AD.TcDUT
{attribute addProperty BoxType "AX8206-0000-0100-0100"}
{attribute addProperty Id "DeviceDevice_F82A60211620Ch_ACh_A_359CD49A176220Ch_BCh_B_71B491C3176220WcStateAT %I*WcState_98A4DF7520.250InfoDataAT %I*InfoData_17277C5A208260"}
{attribute addProperty CRC "2029095651"}
{attribute addProperty SizeInBites "578"}
{attribute addProperty SizeInBytes "72.25"}
TYPE AX8206_06F284AD :
STRUCT
	{attribute addProperty Name "Device"}
	Device : Device_F82A6021;
	{attribute addProperty Name "Ch_A"}
	Ch_A : Ch_A_359CD49A;
	{attribute addProperty Name "Ch_B"}
	Ch_B : Ch_B_71B491C3;
	{attribute addProperty Name "WcState"}
	WcState : WcState_98A4DF75;
	{attribute addProperty Name "InfoData"}
	InfoData : InfoData_17277C5A;
END_STRUCT
END_TYPE

// ---- DUTs/IO/Boxes/AX8206_23A6453C.TcDUT
{attribute addProperty BoxType "AX8206-0000-0102-0102"}
{attribute addProperty Id "DeviceDevice_F82A60211620Ch_ACh_A_B17182A2176220Ch_BCh_B_7239D878176220WcStateAT %I*WcState_98A4DF7520.250InfoDataAT %I*InfoData_17277C5A208260"}
{attribute addProperty CRC "2269547550"}
{attribute addProperty SizeInBites "578"}
{attribute addProperty SizeInBytes "72.25"}
TYPE AX8206_23A6453C :
STRUCT
	{attribute addProperty Name "Device"}
	Device : Device_F82A6021;
	{attribute addProperty Name "Ch_A"}
	Ch_A : Ch_A_B17182A2;
	{attribute addProperty Name "Ch_B"}
	Ch_B : Ch_B_7239D878;
	{attribute addProperty Name "WcState"}
	WcState : WcState_98A4DF75;
	{attribute addProperty Name "InfoData"}
	InfoData : InfoData_17277C5A;
END_STRUCT
END_TYPE

// ---- DUTs/IO/Boxes/AX8206_36A80AF0.TcDUT
{attribute addProperty BoxType "AX8206-0100-0101-0101"}
{attribute addProperty Id "DeviceDevice_F82A60211620Device_SafetyDevice_Safety_AF71BE9D160200Ch_ACh_A_359CD49A176220Ch_BCh_B_71B491C3176220WcStateAT %I*WcState_DC9C971540.50InfoDataAT %I*InfoData_17277C5A208260"}
{attribute addProperty CRC "932077249"}
{attribute addProperty SizeInBites "740"}
{attribute addProperty SizeInBytes "92.5"}
TYPE AX8206_36A80AF0 :
STRUCT
	{attribute addProperty Name "Device"}
	Device : Device_F82A6021;
	{attribute addProperty Name "Device_Safety"}
	Device_Safety : Device_Safety_AF71BE9D;
	{attribute addProperty Name "Ch_A"}
	Ch_A : Ch_A_359CD49A;
	{attribute addProperty Name "Ch_B"}
	Ch_B : Ch_B_71B491C3;
	{attribute addProperty Name "WcState"}
	WcState : WcState_DC9C9715;
	{attribute addProperty Name "InfoData"}
	InfoData : InfoData_17277C5A;
END_STRUCT
END_TYPE

// ---- DUTs/IO/Boxes/AX8206_AF8A8AFA.TcDUT
{attribute addProperty BoxType "AX8206-0100-0102-0102"}
{attribute addProperty Id "DeviceDevice_F82A60211620Device_SafetyDevice_Safety_AF71BE9D160200Ch_ACh_A_B17182A2176220Ch_BCh_B_7239D878176220WcStateAT %I*WcState_DC9C971540.50InfoDataAT %I*InfoData_17277C5A208260"}
{attribute addProperty CRC "4212748236"}
{attribute addProperty SizeInBites "740"}
{attribute addProperty SizeInBytes "92.5"}
TYPE AX8206_AF8A8AFA :
STRUCT
	{attribute addProperty Name "Device"}
	Device : Device_F82A6021;
	{attribute addProperty Name "Device_Safety"}
	Device_Safety : Device_Safety_AF71BE9D;
	{attribute addProperty Name "Ch_A"}
	Ch_A : Ch_A_B17182A2;
	{attribute addProperty Name "Ch_B"}
	Ch_B : Ch_B_7239D878;
	{attribute addProperty Name "WcState"}
	WcState : WcState_DC9C9715;
	{attribute addProperty Name "InfoData"}
	InfoData : InfoData_17277C5A;
END_STRUCT
END_TYPE

// ---- DUTs/IO/Boxes/AX8620_B97EFC74.TcDUT
{attribute addProperty BoxType "AX8620-0000-0026"}
{attribute addProperty Id "PSM_StatuswordAT %I*PSM_Statusword_32E7AA9A1620WcStateAT %I*WcState_98A4DF7520.250InfoDataAT %I*InfoData_0BDED7BF144180"}
{attribute addProperty CRC "231615263"}
{attribute addProperty SizeInBites "162"}
{attribute addProperty SizeInBytes "20.25"}
TYPE AX8620_B97EFC74 :
STRUCT
	{attribute addProperty Name "PSM_Statusword"}
	PSM_Statusword : PSM_Statusword_32E7AA9A;
	{attribute addProperty Name "WcState"}
	WcState : WcState_98A4DF75;
	{attribute addProperty Name "InfoData"}
	InfoData : InfoData_0BDED7BF;
END_STRUCT
END_TYPE

// ---- DUTs/IO/Boxes/AX8620_5470AD24.TcDUT
{attribute addProperty BoxType "AX8620-0000-0027"}
{attribute addProperty Id "PSM_StatuswordAT %I*PSM_Statusword_C154CB391620WcStateAT %I*WcState_98A4DF7520.250InfoDataAT %I*InfoData_0BDED7BF144180"}
{attribute addProperty CRC "2880182750"}
{attribute addProperty SizeInBites "162"}
{attribute addProperty SizeInBytes "20.25"}
TYPE AX8620_5470AD24 :
STRUCT
	{attribute addProperty Name "PSM_Statusword"}
	PSM_Statusword : PSM_Statusword_C154CB39;
	{attribute addProperty Name "WcState"}
	WcState : WcState_98A4DF75;
	{attribute addProperty Name "InfoData"}
	InfoData : InfoData_0BDED7BF;
END_STRUCT
END_TYPE

// ---- DUTs/IO/Boxes/AX8620_4A923142.TcDUT
{attribute addProperty BoxType "AX8620-0000-0029"}
{attribute addProperty Id "PSM_Controlword_for_axisAT %I*PSM_Controlword_for_axis_59B039C11620WcStateAT %I*WcState_98A4DF7520.250InfoDataAT %I*InfoData_0BDED7BF144180"}
{attribute addProperty CRC "4182654517"}
{attribute addProperty SizeInBites "162"}
{attribute addProperty SizeInBytes "20.25"}
TYPE AX8620_4A923142 :
STRUCT
	{attribute addProperty Name "PSM_Controlword_for_axis"}
	PSM_Controlword_for_axis : PSM_Controlword_for_axis_59B039C1;
	{attribute addProperty Name "WcState"}
	WcState : WcState_98A4DF75;
	{attribute addProperty Name "InfoData"}
	InfoData : InfoData_0BDED7BF;
END_STRUCT
END_TYPE

// ---- DUTs/IO/Boxes/AX8620_56141E8A.TcDUT
{attribute addProperty BoxType "AX8620-1000-0026"}
{attribute addProperty Id "PSM_PSM_StatuswordAT %I*PSM_PSM_Statusword_32E7AA9A1620WcStateAT %I*WcState_98A4DF7520.250InfoDataAT %I*InfoData_0BDED7BF144180"}
{attribute addProperty CRC "1082389167"}
{attribute addProperty SizeInBites "162"}
{attribute addProperty SizeInBytes "20.25"}
TYPE AX8620_56141E8A :
STRUCT
	{attribute addProperty Name "PSM_PSM_Statusword"}
	PSM_PSM_Statusword : PSM_PSM_Statusword_32E7AA9A;
	{attribute addProperty Name "WcState"}
	WcState : WcState_98A4DF75;
	{attribute addProperty Name "InfoData"}
	InfoData : InfoData_0BDED7BF;
END_STRUCT
END_TYPE

// ---- DUTs/IO/Boxes/AX8620_BB1A4FDA.TcDUT
{attribute addProperty BoxType "AX8620-1000-0027"}
{attribute addProperty Id "PSM_PSM_StatuswordAT %I*PSM_PSM_Statusword_C154CB391620WcStateAT %I*WcState_98A4DF7520.250InfoDataAT %I*InfoData_0BDED7BF144180"}
{attribute addProperty CRC "3873554542"}
{attribute addProperty SizeInBites "162"}
{attribute addProperty SizeInBytes "20.25"}
TYPE AX8620_BB1A4FDA :
STRUCT
	{attribute addProperty Name "PSM_PSM_Statusword"}
	PSM_PSM_Statusword : PSM_PSM_Statusword_C154CB39;
	{attribute addProperty Name "WcState"}
	WcState : WcState_98A4DF75;
	{attribute addProperty Name "InfoData"}
	InfoData : InfoData_0BDED7BF;
END_STRUCT
END_TYPE

// ---- DUTs/IO/Boxes/AX8640_56141E8A.TcDUT
{attribute addProperty BoxType "AX8640-0000-0026"}
{attribute addProperty Id "PSM_PSM_StatuswordAT %I*PSM_PSM_Statusword_32E7AA9A1620WcStateAT %I*WcState_98A4DF7520.250InfoDataAT %I*InfoData_0BDED7BF144180"}
{attribute addProperty CRC "1082389167"}
{attribute addProperty SizeInBites "162"}
{attribute addProperty SizeInBytes "20.25"}
TYPE AX8640_56141E8A :
STRUCT
	{attribute addProperty Name "PSM_PSM_Statusword"}
	PSM_PSM_Statusword : PSM_PSM_Statusword_32E7AA9A;
	{attribute addProperty Name "WcState"}
	WcState : WcState_98A4DF75;
	{attribute addProperty Name "InfoData"}
	InfoData : InfoData_0BDED7BF;
END_STRUCT
END_TYPE

// ---- DUTs/IO/Boxes/AX8640_BB1A4FDA.TcDUT
{attribute addProperty BoxType "AX8640-0000-0027"}
{attribute addProperty Id "PSM_PSM_StatuswordAT %I*PSM_PSM_Statusword_C154CB391620WcStateAT %I*WcState_98A4DF7520.250InfoDataAT %I*InfoData_0BDED7BF144180"}
{attribute addProperty CRC "3873554542"}
{attribute addProperty SizeInBites "162"}
{attribute addProperty SizeInBytes "20.25"}
TYPE AX8640_BB1A4FDA :
STRUCT
	{attribute addProperty Name "PSM_PSM_Statusword"}
	PSM_PSM_Statusword : PSM_PSM_Statusword_C154CB39;
	{attribute addProperty Name "WcState"}
	WcState : WcState_98A4DF75;
	{attribute addProperty Name "InfoData"}
	InfoData : InfoData_0BDED7BF;
END_STRUCT
END_TYPE

// ---- DUTs/IO/Boxes/AX8640_4A923142.TcDUT
{attribute addProperty BoxType "AX8640-0000-0029"}
{attribute addProperty Id "PSM_Controlword_for_axisAT %I*PSM_Controlword_for_axis_59B039C11620WcStateAT %I*WcState_98A4DF7520.250InfoDataAT %I*InfoData_0BDED7BF144180"}
{attribute addProperty CRC "4182654517"}
{attribute addProperty SizeInBites "162"}
{attribute addProperty SizeInBytes "20.25"}
TYPE AX8640_4A923142 :
STRUCT
	{attribute addProperty Name "PSM_Controlword_for_axis"}
	PSM_Controlword_for_axis : PSM_Controlword_for_axis_59B039C1;
	{attribute addProperty Name "WcState"}
	WcState : WcState_98A4DF75;
	{attribute addProperty Name "InfoData"}
	InfoData : InfoData_0BDED7BF;
END_STRUCT
END_TYPE

// ---- DUTs/IO/Boxes/AX8810_B7ACDB90.TcDUT
{attribute addProperty BoxType "AX8810-0000-0017"}
{attribute addProperty Id "PSM_StatuswordAT %I*PSM_Statusword_B057017B1620WcStateAT %I*WcState_98A4DF7520.250InfoDataAT %I*InfoData_0BDED7BF144180"}
{attribute addProperty CRC "356712783"}
{attribute addProperty SizeInBites "162"}
{attribute addProperty SizeInBytes "20.25"}
TYPE AX8810_B7ACDB90 :
STRUCT
	{attribute addProperty Name "PSM_Statusword"}
	PSM_Statusword : PSM_Statusword_B057017B;
	{attribute addProperty Name "WcState"}
	WcState : WcState_98A4DF75;
	{attribute addProperty Name "InfoData"}
	InfoData : InfoData_0BDED7BF;
END_STRUCT
END_TYPE

// ---- DUTs/IO/Boxes/AX8810_4A923142.TcDUT
{attribute addProperty BoxType "AX8810-0000-0024-0024"}
{attribute addProperty Id "PSM_Controlword_for_axisAT %I*PSM_Controlword_for_axis_59B039C11620WcStateAT %I*WcState_98A4DF7520.250InfoDataAT %I*InfoData_0BDED7BF144180"}
{attribute addProperty CRC "4182654517"}
{attribute addProperty SizeInBites "162"}
{attribute addProperty SizeInBytes "20.25"}
TYPE AX8810_4A923142 :
STRUCT
	{attribute addProperty Name "PSM_Controlword_for_axis"}
	PSM_Controlword_for_axis : PSM_Controlword_for_axis_59B039C1;
	{attribute addProperty Name "WcState"}
	WcState : WcState_98A4DF75;
	{attribute addProperty Name "InfoData"}
	InfoData : InfoData_0BDED7BF;
END_STRUCT
END_TYPE

// ---- DUTs/IO/Boxes/BK1250_4487A81F.TcDUT
{attribute addProperty BoxType "BK1250-0000-0000"}
{attribute addProperty Id "InputsAT %I*Inputs_6F058048000OutputsAT %I*Outputs_9C14F798000WcStateAT %I*WcState_98A4DF7520.250InfoDataAT %I*InfoData_275E3363128160"}
{attribute addProperty CRC "1783375152"}
{attribute addProperty SizeInBites "130"}
{attribute addProperty SizeInBytes "16.25"}
TYPE BK1250_4487A81F :
STRUCT
	{attribute addProperty Name "Inputs"}
	Inputs : Inputs_6F058048;
	{attribute addProperty Name "Outputs"}
	Outputs : Outputs_9C14F798;
	{attribute addProperty Name "WcState"}
	WcState : WcState_98A4DF75;
	{attribute addProperty Name "InfoData"}
	InfoData : InfoData_275E3363;
END_STRUCT
END_TYPE

// ---- DUTs/IO/Boxes/BK1120_D3F02A0D.TcDUT
{attribute addProperty BoxType "BK1120-0000-0000"}
{attribute addProperty Id "InputsAT %I*Inputs_6F058048000OutputsAT %I*Outputs_9C14F798000WcStateAT %I*WcState_98A4DF7520.250InfoDataAT %I*InfoData_BC63D37F80100"}
{attribute addProperty CRC "2670801399"}
{attribute addProperty SizeInBites "82"}
{attribute addProperty SizeInBytes "10.25"}
TYPE BK1120_D3F02A0D :
STRUCT
	{attribute addProperty Name "Inputs"}
	Inputs : Inputs_6F058048;
	{attribute addProperty Name "Outputs"}
	Outputs : Outputs_9C14F798;
	{attribute addProperty Name "WcState"}
	WcState : WcState_98A4DF75;
	{attribute addProperty Name "InfoData"}
	InfoData : InfoData_BC63D37F;
END_STRUCT
END_TYPE

// ---- DUTs/IO/Boxes/BK1120_4487A81F.TcDUT
{attribute addProperty BoxType "BK1120-0000-0001"}
{attribute addProperty Id "InputsAT %I*Inputs_6F058048000OutputsAT %I*Outputs_9C14F798000WcStateAT %I*WcState_98A4DF7520.250InfoDataAT %I*InfoData_275E3363128160"}
{attribute addProperty CRC "1783375152"}
{attribute addProperty SizeInBites "130"}
{attribute addProperty SizeInBytes "16.25"}
TYPE BK1120_4487A81F :
STRUCT
	{attribute addProperty Name "Inputs"}
	Inputs : Inputs_6F058048;
	{attribute addProperty Name "Outputs"}
	Outputs : Outputs_9C14F798;
	{attribute addProperty Name "WcState"}
	WcState : WcState_98A4DF75;
	{attribute addProperty Name "InfoData"}
	InfoData : InfoData_275E3363;
END_STRUCT
END_TYPE

// ---- DUTs/IO/Boxes/CPXXXX_4487A81F.TcDUT
{attribute addProperty BoxType "CPXXXX-BK7902-0016"}
{attribute addProperty Id "InputsAT %I*Inputs_6F058048000OutputsAT %I*Outputs_9C14F798000WcStateAT %I*WcState_98A4DF7520.250InfoDataAT %I*InfoData_275E3363128160"}
{attribute addProperty CRC "1783375152"}
{attribute addProperty SizeInBites "130"}
{attribute addProperty SizeInBytes "16.25"}
TYPE CPXXXX_4487A81F :
STRUCT
	{attribute addProperty Name "Inputs"}
	Inputs : Inputs_6F058048;
	{attribute addProperty Name "Outputs"}
	Outputs : Outputs_9C14F798;
	{attribute addProperty Name "WcState"}
	WcState : WcState_98A4DF75;
	{attribute addProperty Name "InfoData"}
	InfoData : InfoData_275E3363;
END_STRUCT
END_TYPE

// ---- DUTs/IO/Boxes/BK1150_4487A81F.TcDUT
{attribute addProperty BoxType "BK1150-0000-0016"}
{attribute addProperty Id "InputsAT %I*Inputs_6F058048000OutputsAT %I*Outputs_9C14F798000WcStateAT %I*WcState_98A4DF7520.250InfoDataAT %I*InfoData_275E3363128160"}
{attribute addProperty CRC "1783375152"}
{attribute addProperty SizeInBites "130"}
{attribute addProperty SizeInBytes "16.25"}
TYPE BK1150_4487A81F :
STRUCT
	{attribute addProperty Name "Inputs"}
	Inputs : Inputs_6F058048;
	{attribute addProperty Name "Outputs"}
	Outputs : Outputs_9C14F798;
	{attribute addProperty Name "WcState"}
	WcState : WcState_98A4DF75;
	{attribute addProperty Name "InfoData"}
	InfoData : InfoData_275E3363;
END_STRUCT
END_TYPE

// ---- DUTs/IO/Boxes/CU1123_179A0949.TcDUT
{attribute addProperty BoxType "CU1123-0000-0016"}
{attribute addProperty Id "InfoDataInfoData_192954DE162"}
{attribute addProperty CRC "395970889"}
{attribute addProperty SizeInBites "16"}
{attribute addProperty SizeInBytes "2"}
TYPE CU1123_179A0949 :
STRUCT
	{attribute addProperty Name "InfoData"}
	InfoData : InfoData_192954DE;
END_STRUCT
END_TYPE

// ---- DUTs/IO/Boxes/CU1124_179A0949.TcDUT
{attribute addProperty BoxType "CU1124-0000-0016"}
{attribute addProperty Id "InfoDataInfoData_192954DE162"}
{attribute addProperty CRC "395970889"}
{attribute addProperty SizeInBites "16"}
{attribute addProperty SizeInBytes "2"}
TYPE CU1124_179A0949 :
STRUCT
	{attribute addProperty Name "InfoData"}
	InfoData : InfoData_192954DE;
END_STRUCT
END_TYPE

// ---- DUTs/IO/Boxes/CU1128_179A0949.TcDUT
{attribute addProperty BoxType "CU1128--0000"}
{attribute addProperty Id "InfoDataInfoData_192954DE162"}
{attribute addProperty CRC "395970889"}
{attribute addProperty SizeInBites "16"}
{attribute addProperty SizeInBytes "2"}
TYPE CU1128_179A0949 :
STRUCT
	{attribute addProperty Name "InfoData"}
	InfoData : InfoData_192954DE;
END_STRUCT
END_TYPE

// ---- DUTs/IO/Boxes/CU1521_179A0949.TcDUT
{attribute addProperty BoxType "CU1521-0010-0000"}
{attribute addProperty Id "InfoDataInfoData_192954DE162"}
{attribute addProperty CRC "395970889"}
{attribute addProperty SizeInBites "16"}
{attribute addProperty SizeInBytes "2"}
TYPE CU1521_179A0949 :
STRUCT
	{attribute addProperty Name "InfoData"}
	InfoData : InfoData_192954DE;
END_STRUCT
END_TYPE

// ---- DUTs/IO/Boxes/CU1561_179A0949.TcDUT
{attribute addProperty BoxType "CU1561--0000"}
{attribute addProperty Id "InfoDataInfoData_192954DE162"}
{attribute addProperty CRC "395970889"}
{attribute addProperty SizeInBites "16"}
{attribute addProperty SizeInBytes "2"}
TYPE CU1561_179A0949 :
STRUCT
	{attribute addProperty Name "InfoData"}
	InfoData : InfoData_192954DE;
END_STRUCT
END_TYPE

// ---- DUTs/IO/Boxes/CU2508_179A0949.TcDUT
{attribute addProperty BoxType "CU2508--0000"}
{attribute addProperty Id "InfoDataInfoData_192954DE162"}
{attribute addProperty CRC "395970889"}
{attribute addProperty SizeInBites "16"}
{attribute addProperty SizeInBytes "2"}
TYPE CU2508_179A0949 :
STRUCT
	{attribute addProperty Name "InfoData"}
	InfoData : InfoData_192954DE;
END_STRUCT
END_TYPE

// ---- DUTs/IO/Boxes/CU2508_194A340D.TcDUT
{attribute addProperty BoxType "CU2508-0000-0016"}
{attribute addProperty Id "InfoDataInfoData_BC63D37F8010"}
{attribute addProperty CRC "424293389"}
{attribute addProperty SizeInBites "80"}
{attribute addProperty SizeInBytes "10"}
TYPE CU2508_194A340D :
STRUCT
	{attribute addProperty Name "InfoData"}
	InfoData : InfoData_BC63D37F;
END_STRUCT
END_TYPE

// ---- DUTs/IO/Boxes/CU2508_36DE2952.TcDUT
{attribute addProperty BoxType "CU2508-0000-0017"}
{attribute addProperty Id "EPM_Inputs_ChannelAT %I*ARRAY[0..18] OF EPM_Inputs_Channel_7B63A807160200WcStateAT %I*WcState_98A4DF7520.250InfoDataAT %I*InfoData_BC63D37F80100"}
{attribute addProperty CRC "2816817870"}
{attribute addProperty SizeInBites "242"}
{attribute addProperty SizeInBytes "30.25"}
TYPE CU2508_36DE2952 :
STRUCT
	{attribute addProperty Name "EPM_Inputs_Channel"}
	EPM_Inputs_Channel : ARRAY[0..18] OF EPM_Inputs_Channel_7B63A807;
	{attribute addProperty Name "WcState"}
	WcState : WcState_98A4DF75;
	{attribute addProperty Name "InfoData"}
	InfoData : InfoData_BC63D37F;
END_STRUCT
END_TYPE

// ---- DUTs/IO/Boxes/CX1100_179A0949.TcDUT
{attribute addProperty BoxType "CX1100-0004-0000"}
{attribute addProperty Id "InfoDataInfoData_192954DE162"}
{attribute addProperty CRC "395970889"}
{attribute addProperty SizeInBites "16"}
{attribute addProperty SizeInBytes "2"}
TYPE CX1100_179A0949 :
STRUCT
	{attribute addProperty Name "InfoData"}
	InfoData : InfoData_192954DE;
END_STRUCT
END_TYPE

// ---- DUTs/IO/Boxes/CX5010_EtherCAT_slave_16898E41.TcDUT
{attribute addProperty BoxType "CX5010 EtherCAT slave-1b82-0016"}
{attribute addProperty Id "IO_InputsEMPTY_STRUCTURE000Device_Status_MappingAT %I*Device_Status_Mapping_AC515E2C1620IO_OutputsEMPTY_STRUCTURE000WcStateAT %I*WcState_98A4DF7520.250InfoDataAT %I*InfoData_275E3363128160"}
{attribute addProperty CRC "257024818"}
{attribute addProperty SizeInBites "146"}
{attribute addProperty SizeInBytes "18.25"}
TYPE CX5010_EtherCAT_slave_16898E41 :
STRUCT
	{attribute addProperty Name "IO_Inputs"}
	IO_Inputs : EMPTY_STRUCTURE;
	{attribute addProperty Name "Device_Status_Mapping"}
	Device_Status_Mapping : Device_Status_Mapping_AC515E2C;
	{attribute addProperty Name "IO_Outputs"}
	IO_Outputs : EMPTY_STRUCTURE;
	{attribute addProperty Name "WcState"}
	WcState : WcState_98A4DF75;
	{attribute addProperty Name "InfoData"}
	InfoData : InfoData_275E3363;
END_STRUCT
END_TYPE

// ---- DUTs/IO/Boxes/CX5020_EtherCAT_slave_16898E41.TcDUT
{attribute addProperty BoxType "CX5020 EtherCAT slave-1b82-0016"}
{attribute addProperty Id "IO_InputsEMPTY_STRUCTURE000Device_Status_MappingAT %I*Device_Status_Mapping_AC515E2C1620IO_OutputsEMPTY_STRUCTURE000WcStateAT %I*WcState_98A4DF7520.250InfoDataAT %I*InfoData_275E3363128160"}
{attribute addProperty CRC "257024818"}
{attribute addProperty SizeInBites "146"}
{attribute addProperty SizeInBytes "18.25"}
TYPE CX5020_EtherCAT_slave_16898E41 :
STRUCT
	{attribute addProperty Name "IO_Inputs"}
	IO_Inputs : EMPTY_STRUCTURE;
	{attribute addProperty Name "Device_Status_Mapping"}
	Device_Status_Mapping : Device_Status_Mapping_AC515E2C;
	{attribute addProperty Name "IO_Outputs"}
	IO_Outputs : EMPTY_STRUCTURE;
	{attribute addProperty Name "WcState"}
	WcState : WcState_98A4DF75;
	{attribute addProperty Name "InfoData"}
	InfoData : InfoData_275E3363;
END_STRUCT
END_TYPE

// ---- DUTs/IO/Boxes/CX8010_EtherCAT_slave_16898E41.TcDUT
{attribute addProperty BoxType "CX8010 EtherCAT slave-0000-0016"}
{attribute addProperty Id "IO_InputsEMPTY_STRUCTURE000Device_Status_MappingAT %I*Device_Status_Mapping_AC515E2C1620IO_OutputsEMPTY_STRUCTURE000WcStateAT %I*WcState_98A4DF7520.250InfoDataAT %I*InfoData_275E3363128160"}
{attribute addProperty CRC "257024818"}
{attribute addProperty SizeInBites "146"}
{attribute addProperty SizeInBytes "18.25"}
TYPE CX8010_EtherCAT_slave_16898E41 :
STRUCT
	{attribute addProperty Name "IO_Inputs"}
	IO_Inputs : EMPTY_STRUCTURE;
	{attribute addProperty Name "Device_Status_Mapping"}
	Device_Status_Mapping : Device_Status_Mapping_AC515E2C;
	{attribute addProperty Name "IO_Outputs"}
	IO_Outputs : EMPTY_STRUCTURE;
	{attribute addProperty Name "WcState"}
	WcState : WcState_98A4DF75;
	{attribute addProperty Name "InfoData"}
	InfoData : InfoData_275E3363;
END_STRUCT
END_TYPE

// ---- DUTs/IO/Boxes/CX8110_EtherCAT_slave_16898E41.TcDUT
{attribute addProperty BoxType "CX8110 EtherCAT slave-0000-0016"}
{attribute addProperty Id "IO_InputsEMPTY_STRUCTURE000Device_Status_MappingAT %I*Device_Status_Mapping_AC515E2C1620IO_OutputsEMPTY_STRUCTURE000WcStateAT %I*WcState_98A4DF7520.250InfoDataAT %I*InfoData_275E3363128160"}
{attribute addProperty CRC "257024818"}
{attribute addProperty SizeInBites "146"}
{attribute addProperty SizeInBytes "18.25"}
TYPE CX8110_EtherCAT_slave_16898E41 :
STRUCT
	{attribute addProperty Name "IO_Inputs"}
	IO_Inputs : EMPTY_STRUCTURE;
	{attribute addProperty Name "Device_Status_Mapping"}
	Device_Status_Mapping : Device_Status_Mapping_AC515E2C;
	{attribute addProperty Name "IO_Outputs"}
	IO_Outputs : EMPTY_STRUCTURE;
	{attribute addProperty Name "WcState"}
	WcState : WcState_98A4DF75;
	{attribute addProperty Name "InfoData"}
	InfoData : InfoData_275E3363;
END_STRUCT
END_TYPE

// ---- DUTs/IO/Boxes/CX2020_EtherCAT_slave_16898E41.TcDUT
{attribute addProperty BoxType "CX2020 EtherCAT slave-1b82-0016"}
{attribute addProperty Id "IO_InputsEMPTY_STRUCTURE000Device_Status_MappingAT %I*Device_Status_Mapping_AC515E2C1620IO_OutputsEMPTY_STRUCTURE000WcStateAT %I*WcState_98A4DF7520.250InfoDataAT %I*InfoData_275E3363128160"}
{attribute addProperty CRC "257024818"}
{attribute addProperty SizeInBites "146"}
{attribute addProperty SizeInBytes "18.25"}
TYPE CX2020_EtherCAT_slave_16898E41 :
STRUCT
	{attribute addProperty Name "IO_Inputs"}
	IO_Inputs : EMPTY_STRUCTURE;
	{attribute addProperty Name "Device_Status_Mapping"}
	Device_Status_Mapping : Device_Status_Mapping_AC515E2C;
	{attribute addProperty Name "IO_Outputs"}
	IO_Outputs : EMPTY_STRUCTURE;
	{attribute addProperty Name "WcState"}
	WcState : WcState_98A4DF75;
	{attribute addProperty Name "InfoData"}
	InfoData : InfoData_275E3363;
END_STRUCT
END_TYPE

// ---- DUTs/IO/Boxes/CX2030_EtherCAT_slave_16898E41.TcDUT
{attribute addProperty BoxType "CX2030 EtherCAT slave-1b82-0016"}
{attribute addProperty Id "IO_InputsEMPTY_STRUCTURE000Device_Status_MappingAT %I*Device_Status_Mapping_AC515E2C1620IO_OutputsEMPTY_STRUCTURE000WcStateAT %I*WcState_98A4DF7520.250InfoDataAT %I*InfoData_275E3363128160"}
{attribute addProperty CRC "257024818"}
{attribute addProperty SizeInBites "146"}
{attribute addProperty SizeInBytes "18.25"}
TYPE CX2030_EtherCAT_slave_16898E41 :
STRUCT
	{attribute addProperty Name "IO_Inputs"}
	IO_Inputs : EMPTY_STRUCTURE;
	{attribute addProperty Name "Device_Status_Mapping"}
	Device_Status_Mapping : Device_Status_Mapping_AC515E2C;
	{attribute addProperty Name "IO_Outputs"}
	IO_Outputs : EMPTY_STRUCTURE;
	{attribute addProperty Name "WcState"}
	WcState : WcState_98A4DF75;
	{attribute addProperty Name "InfoData"}
	InfoData : InfoData_275E3363;
END_STRUCT
END_TYPE

// ---- DUTs/IO/Boxes/CX2033_EtherCAT_slave_16898E41.TcDUT
{attribute addProperty BoxType "CX2033 EtherCAT slave-1b82-0016"}
{attribute addProperty Id "IO_InputsEMPTY_STRUCTURE000Device_Status_MappingAT %I*Device_Status_Mapping_AC515E2C1620IO_OutputsEMPTY_STRUCTURE000WcStateAT %I*WcState_98A4DF7520.250InfoDataAT %I*InfoData_275E3363128160"}
{attribute addProperty CRC "257024818"}
{attribute addProperty SizeInBites "146"}
{attribute addProperty SizeInBytes "18.25"}
TYPE CX2033_EtherCAT_slave_16898E41 :
STRUCT
	{attribute addProperty Name "IO_Inputs"}
	IO_Inputs : EMPTY_STRUCTURE;
	{attribute addProperty Name "Device_Status_Mapping"}
	Device_Status_Mapping : Device_Status_Mapping_AC515E2C;
	{attribute addProperty Name "IO_Outputs"}
	IO_Outputs : EMPTY_STRUCTURE;
	{attribute addProperty Name "WcState"}
	WcState : WcState_98A4DF75;
	{attribute addProperty Name "InfoData"}
	InfoData : InfoData_275E3363;
END_STRUCT
END_TYPE

// ---- DUTs/IO/Boxes/CX2040_EtherCAT_slave_16898E41.TcDUT
{attribute addProperty BoxType "CX2040 EtherCAT slave-1b82-0016"}
{attribute addProperty Id "IO_InputsEMPTY_STRUCTURE000Device_Status_MappingAT %I*Device_Status_Mapping_AC515E2C1620IO_OutputsEMPTY_STRUCTURE000WcStateAT %I*WcState_98A4DF7520.250InfoDataAT %I*InfoData_275E3363128160"}
{attribute addProperty CRC "257024818"}
{attribute addProperty SizeInBites "146"}
{attribute addProperty SizeInBytes "18.25"}
TYPE CX2040_EtherCAT_slave_16898E41 :
STRUCT
	{attribute addProperty Name "IO_Inputs"}
	IO_Inputs : EMPTY_STRUCTURE;
	{attribute addProperty Name "Device_Status_Mapping"}
	Device_Status_Mapping : Device_Status_Mapping_AC515E2C;
	{attribute addProperty Name "IO_Outputs"}
	IO_Outputs : EMPTY_STRUCTURE;
	{attribute addProperty Name "WcState"}
	WcState : WcState_98A4DF75;
	{attribute addProperty Name "InfoData"}
	InfoData : InfoData_275E3363;
END_STRUCT
END_TYPE

// ---- DUTs/IO/Boxes/CX2042_EtherCAT_slave_16898E41.TcDUT
{attribute addProperty BoxType "CX2042 EtherCAT slave-1b82-0016"}
{attribute addProperty Id "IO_InputsEMPTY_STRUCTURE000Device_Status_MappingAT %I*Device_Status_Mapping_AC515E2C1620IO_OutputsEMPTY_STRUCTURE000WcStateAT %I*WcState_98A4DF7520.250InfoDataAT %I*InfoData_275E3363128160"}
{attribute addProperty CRC "257024818"}
{attribute addProperty SizeInBites "146"}
{attribute addProperty SizeInBytes "18.25"}
TYPE CX2042_EtherCAT_slave_16898E41 :
STRUCT
	{attribute addProperty Name "IO_Inputs"}
	IO_Inputs : EMPTY_STRUCTURE;
	{attribute addProperty Name "Device_Status_Mapping"}
	Device_Status_Mapping : Device_Status_Mapping_AC515E2C;
	{attribute addProperty Name "IO_Outputs"}
	IO_Outputs : EMPTY_STRUCTURE;
	{attribute addProperty Name "WcState"}
	WcState : WcState_98A4DF75;
	{attribute addProperty Name "InfoData"}
	InfoData : InfoData_275E3363;
END_STRUCT
END_TYPE

// ---- DUTs/IO/Boxes/CX2043_EtherCAT_slave_16898E41.TcDUT
{attribute addProperty BoxType "CX2043 EtherCAT slave-1b82-0016"}
{attribute addProperty Id "IO_InputsEMPTY_STRUCTURE000Device_Status_MappingAT %I*Device_Status_Mapping_AC515E2C1620IO_OutputsEMPTY_STRUCTURE000WcStateAT %I*WcState_98A4DF7520.250InfoDataAT %I*InfoData_275E3363128160"}
{attribute addProperty CRC "257024818"}
{attribute addProperty SizeInBites "146"}
{attribute addProperty SizeInBytes "18.25"}
TYPE CX2043_EtherCAT_slave_16898E41 :
STRUCT
	{attribute addProperty Name "IO_Inputs"}
	IO_Inputs : EMPTY_STRUCTURE;
	{attribute addProperty Name "Device_Status_Mapping"}
	Device_Status_Mapping : Device_Status_Mapping_AC515E2C;
	{attribute addProperty Name "IO_Outputs"}
	IO_Outputs : EMPTY_STRUCTURE;
	{attribute addProperty Name "WcState"}
	WcState : WcState_98A4DF75;
	{attribute addProperty Name "InfoData"}
	InfoData : InfoData_275E3363;
END_STRUCT
END_TYPE

// ---- DUTs/IO/Boxes/CX2062_EtherCAT_slave_16898E41.TcDUT
{attribute addProperty BoxType "CX2062 EtherCAT slave-1b82-0016"}
{attribute addProperty Id "IO_InputsEMPTY_STRUCTURE000Device_Status_MappingAT %I*Device_Status_Mapping_AC515E2C1620IO_OutputsEMPTY_STRUCTURE000WcStateAT %I*WcState_98A4DF7520.250InfoDataAT %I*InfoData_275E3363128160"}
{attribute addProperty CRC "257024818"}
{attribute addProperty SizeInBites "146"}
{attribute addProperty SizeInBytes "18.25"}
TYPE CX2062_EtherCAT_slave_16898E41 :
STRUCT
	{attribute addProperty Name "IO_Inputs"}
	IO_Inputs : EMPTY_STRUCTURE;
	{attribute addProperty Name "Device_Status_Mapping"}
	Device_Status_Mapping : Device_Status_Mapping_AC515E2C;
	{attribute addProperty Name "IO_Outputs"}
	IO_Outputs : EMPTY_STRUCTURE;
	{attribute addProperty Name "WcState"}
	WcState : WcState_98A4DF75;
	{attribute addProperty Name "InfoData"}
	InfoData : InfoData_275E3363;
END_STRUCT
END_TYPE

